C05484=1159.345,41.172,-49.319,-179.753,6.177,149.041
C05485=1159.351,40.923,-49.303,-179.756,6.176,149.042
C05486=1159.355,40.674,-49.288,-179.758,6.176,149.043
C05487=1159.361,40.424,-49.273,-179.761,6.174,149.043
C05488=1159.365,40.174,-49.258,-179.763,6.173,149.044
C05489=1159.371,39.924,-49.242,-179.766,6.173,149.044
C05490=1159.375,39.675,-49.227,-179.769,6.171,149.045
C05491=1159.381,39.425,-49.212,-179.771,6.171,149.045
C05492=1159.386,39.176,-49.198,-179.774,6.170,149.046
C05493=1159.391,38.927,-49.182,-179.777,6.169,149.047
C05494=1159.396,38.678,-49.167,-179.779,6.168,149.047
C05495=1159.401,38.428,-49.152,-179.782,6.167,149.048
C05496=1159.405,38.178,-49.137,-179.784,6.166,149.048
C05497=1159.411,37.928,-49.121,-179.787,6.165,149.049
C05498=1159.415,37.679,-49.106,-179.789,6.164,149.049
C05499=1159.421,37.429,-49.091,-179.792,6.163,149.050
C05500=1159.426,37.180,-49.076,-179.795,6.162,149.050
C05501=1159.431,36.931,-49.061,-179.797,6.162,149.051
C05502=1159.436,36.681,-49.046,-179.800,6.160,149.052
C05503=1159.441,36.432,-49.031,-179.803,6.160,149.052
C05504=1159.446,36.183,-49.016,-179.805,6.159,149.053
C05505=1159.452,35.933,-49.001,-179.807,6.158,149.053
C05506=1159.456,35.684,-48.986,-179.810,6.157,149.054
C05507=1159.462,35.434,-48.970,-179.813,6.156,149.054
C05508=1159.466,35.184,-48.956,-179.815,6.155,149.055
C05509=1159.471,34.935,-48.941,-179.818,6.154,149.056
C05510=1159.477,34.685,-48.926,-179.820,6.153,149.056
C05511=1159.481,34.436,-48.911,-179.823,6.153,149.057
C05512=1159.487,34.186,-48.895,-179.826,6.151,149.057
C05513=1159.491,33.936,-48.881,-179.828,6.151,149.058
C05514=1159.496,33.687,-48.866,-179.831,6.150,149.058
C05515=1159.502,33.437,-48.851,-179.834,6.148,149.059
C05516=1159.506,33.188,-48.836,-179.836,6.148,149.059
C05517=1159.511,32.939,-48.822,-179.839,6.147,149.060
C05518=1159.517,32.689,-48.806,-179.841,6.146,149.061
C05519=1159.522,32.439,-48.792,-179.844,6.145,149.061
C05520=1159.526,32.190,-48.777,-179.846,6.144,149.062
C05521=1159.532,31.941,-48.761,-179.849,6.144,149.062
C05522=1159.537,31.691,-48.747,-179.852,6.142,149.063
C05523=1159.542,31.441,-48.733,-179.854,6.142,149.063
C05524=1159.547,31.192,-48.717,-179.856,6.141,149.064
C05525=1159.552,30.942,-48.703,-179.859,6.140,149.065
C05526=1159.557,30.693,-48.688,-179.862,6.139,149.065
C05527=1159.562,30.443,-48.673,-179.864,6.138,149.066
C05528=1159.567,30.194,-48.658,-179.867,6.137,149.066
C05529=1159.572,29.944,-48.644,-179.870,6.136,149.067
C05530=1159.577,29.695,-48.628,-179.872,6.135,149.067
C05531=1159.582,29.445,-48.614,-179.875,6.135,149.068
C05532=1159.587,29.196,-48.600,-179.877,6.134,149.068
C05533=1159.592,28.947,-48.585,-179.880,6.133,149.069
C05534=1159.598,28.697,-48.570,-179.882,6.132,149.070
C05535=1159.602,28.447,-48.555,-179.885,6.131,149.070
C05536=1159.608,28.178,-48.540,-179.888,6.130,149.071
C05537=1159.613,27.910,-48.525,-179.890,6.129,149.071
C05538=1159.619,27.641,-48.508,-179.893,6.129,149.072
C05539=1159.624,27.372,-48.493,-179.896,6.127,149.073
C05540=1159.629,27.122,-48.478,-179.898,6.127,149.073
C05541=1159.635,26.873,-48.463,-179.901,6.126,149.074
C05542=1159.640,26.623,-48.448,-179.904,6.125,149.074
C05543=1159.645,26.373,-48.434,-179.906,6.124,149.075
C05544=1159.649,26.124,-48.419,-179.909,6.123,149.075
C05545=1159.654,25.875,-48.405,-179.911,6.123,149.076
C05546=1159.659,25.625,-48.391,-179.914,6.121,149.077
C05547=1159.665,25.375,-48.376,-179.917,6.121,149.077
C05548=1159.670,25.127,-48.361,-179.919,6.120,149.078
C05549=1159.675,24.877,-48.347,-179.921,6.119,149.078
C05550=1159.680,24.627,-48.332,-179.924,6.118,149.079
C05551=1159.685,24.377,-48.318,-179.927,6.117,149.080
C05552=1159.690,24.128,-48.303,-179.929,6.116,149.080
C05553=1159.695,23.878,-48.288,-179.932,6.116,149.081
C05554=1159.700,23.629,-48.274,-179.934,6.114,149.081
C05555=1159.705,23.379,-48.260,-179.937,6.114,149.082
C05556=1159.711,23.130,-48.246,-179.939,6.113,149.082
C05557=1159.716,22.881,-48.231,-179.942,6.112,149.083
C05558=1159.720,22.631,-48.217,-179.945,6.111,149.083
C05559=1159.725,22.381,-48.202,-179.947,6.110,149.084
C05560=1159.730,22.132,-48.188,-179.949,6.110,149.084
C05561=1159.735,21.882,-48.174,-179.952,6.109,149.085
C05562=1159.741,21.633,-48.160,-179.954,6.108,149.086
C05563=1159.746,21.384,-48.144,-179.958,6.107,149.086
C05564=1159.751,21.134,-48.130,-179.960,6.106,149.087
C05565=1159.756,20.884,-48.116,-179.962,6.106,149.087
C05566=1159.761,20.634,-48.101,-179.964,6.105,149.088
C05567=1159.766,20.385,-48.087,-179.968,6.104,149.089
C05568=1159.772,20.136,-48.073,-179.970,6.103,149.089
C05569=1159.777,19.886,-48.059,-179.973,6.102,149.090
C05570=1159.782,19.636,-48.045,-179.975,6.102,149.090
C05571=1159.787,19.387,-48.030,-179.977,6.101,149.091
C05572=1159.791,19.137,-48.016,-179.981,6.100,149.092
C05573=1159.797,18.888,-48.002,-179.983,6.099,149.092
C05574=1159.802,18.638,-47.988,-179.985,6.098,149.093
C05575=1159.807,18.388,-47.974,-179.988,6.098,149.093
C05576=1159.812,18.139,-47.959,-179.990,6.097,149.094
C05577=1159.817,17.889,-47.945,-179.993,6.095,149.094
C05578=1159.822,17.640,-47.931,-179.996,6.095,149.095
C05579=1159.827,17.390,-47.917,-179.998,6.094,149.095
C05580=1159.832,17.141,-47.903,180.000,6.094,149.096
C05581=1159.837,16.891,-47.888,179.997,6.093,149.097
C05582=1159.843,16.642,-47.874,179.994,6.092,149.097
C05583=1159.848,16.392,-47.860,179.992,6.091,149.098
C05584=1159.853,16.142,-47.846,179.989,6.090,149.098
C05585=1159.858,15.893,-47.832,179.987,6.089,149.099
C05586=1159.863,15.644,-47.818,179.984,6.089,149.100
C05587=1159.867,15.394,-47.804,179.981,6.088,149.100
C05588=1159.872,15.145,-47.790,179.979,6.087,149.101
C05589=1159.878,14.896,-47.776,179.976,6.086,149.101
C05590=1159.883,14.646,-47.762,179.974,6.086,149.102
C05591=1159.888,14.396,-47.748,179.972,6.085,149.102
C05592=1159.893,14.146,-47.734,179.969,6.084,149.103
C05593=1159.899,13.897,-47.720,179.966,6.083,149.104
C05594=1159.904,13.647,-47.706,179.964,6.082,149.104
C05595=1159.909,13.397,-47.691,179.961,6.082,149.105
C05596=1159.913,13.149,-47.678,179.959,6.081,149.105
C05597=1159.918,12.899,-47.664,179.957,6.080,149.106
C05598=1159.924,12.649,-47.650,179.954,6.079,149.106
C05599=1159.929,12.400,-47.636,179.951,6.078,149.107
C05600=1159.934,12.150,-47.622,179.949,6.078,149.108
C05601=1159.939,11.900,-47.608,179.946,6.077,149.108
C05602=1159.943,11.651,-47.594,179.944,6.076,149.109
C05603=1159.949,11.401,-47.581,179.942,6.076,149.109
C05604=1159.954,11.152,-47.567,179.938,6.075,149.110
C05605=1159.960,10.903,-47.553,179.936,6.074,149.110
C05606=1159.965,10.653,-47.538,179.933,6.073,149.111
C05607=1159.970,10.402,-47.525,179.931,6.072,149.112
C05608=1159.975,10.154,-47.511,179.929,6.072,149.112
C05609=1159.980,9.904,-47.497,179.926,6.071,149.113
C05610=1159.985,9.654,-47.483,179.924,6.071,149.113
C05611=1159.991,9.405,-47.470,179.921,6.069,149.114
C05612=1159.995,9.155,-47.456,179.918,6.069,149.115
C05613=1160.000,8.906,-47.442,179.916,6.068,149.115
C05614=1160.006,8.656,-47.429,179.914,6.067,149.116
C05615=1160.010,8.406,-47.414,179.911,6.066,149.116
C05616=1160.015,8.158,-47.401,179.909,6.066,149.117
C05617=1160.021,7.907,-47.387,179.906,6.066,149.118
C05618=1160.026,7.658,-47.373,179.903,6.064,149.118
C05619=1160.031,7.409,-47.359,179.901,6.064,149.119
C05620=1160.036,7.158,-47.346,179.898,6.063,149.119
C05621=1160.041,6.909,-47.332,179.896,6.062,149.120
C05622=1160.046,6.659,-47.319,179.894,6.061,149.120
C05623=1160.051,6.409,-47.304,179.891,6.061,149.121
C05624=1160.056,6.161,-47.291,179.889,6.060,149.121
C05625=1160.061,5.910,-47.278,179.886,6.059,149.122
C05626=1160.067,5.661,-47.264,179.883,6.058,149.123
C05627=1160.072,5.411,-47.251,179.881,6.058,149.123
C05628=1160.076,5.162,-47.236,179.879,6.057,149.124
C05629=1160.082,4.913,-47.223,179.876,6.056,149.124
C05630=1160.087,4.663,-47.210,179.873,6.056,149.125
C05631=1160.092,4.414,-47.196,179.871,6.055,149.126
C05632=1160.097,4.163,-47.182,179.868,6.055,149.126
C05633=1160.102,3.915,-47.169,179.866,6.053,149.127
C05634=1160.107,3.664,-47.155,179.863,6.052,149.127
C05635=1160.112,3.416,-47.142,179.861,6.052,149.128
C05636=1160.118,3.165,-47.128,179.858,6.051,149.129
C05637=1160.123,2.916,-47.114,179.856,6.050,149.129
C05638=1160.128,2.666,-47.101,179.853,6.050,149.130
C05639=1160.133,2.417,-47.087,179.851,6.049,149.130
C05640=1160.139,2.147,-47.073,179.849,6.049,149.131
C05641=1160.144,1.878,-47.059,179.845,6.047,149.132
C05642=1160.149,1.609,-47.044,179.843,6.047,149.132
C05643=1160.155,1.339,-47.030,179.840,6.046,149.133
C05644=1160.160,1.090,-47.016,179.838,6.046,149.133
C05645=1160.165,0.840,-47.003,179.836,6.045,149.134
C05646=1160.170,0.591,-46.989,179.832,6.044,149.135
C05647=1160.176,0.341,-46.976,179.830,6.043,149.135
C05648=1160.181,0.091,-46.963,179.828,6.042,149.136
C05649=1160.186,-0.158,-46.949,179.825,6.042,149.136
C05650=1160.191,-0.408,-46.936,179.823,6.041,149.137
C05651=1160.196,-0.657,-46.923,179.820,6.041,149.138
C05652=1160.201,-0.907,-46.909,179.818,6.040,149.138
C05653=1160.207,-1.157,-46.896,179.815,6.039,149.139
C05654=1160.211,-1.407,-46.883,179.813,6.039,149.139
C05655=1160.217,-1.656,-46.869,179.810,6.038,149.140
C05656=1160.221,-1.906,-46.856,179.808,6.037,149.140
C05657=1160.227,-2.155,-46.843,179.805,6.036,149.141
C05658=1160.231,-2.405,-46.829,179.802,6.036,149.142
C05659=1160.237,-2.654,-46.816,179.800,6.035,149.142
C05660=1160.242,-2.904,-46.803,179.798,6.034,149.143
C05661=1160.247,-3.153,-46.789,179.795,6.033,149.143
C05662=1160.253,-3.403,-46.776,179.793,6.033,149.144
C05663=1160.257,-3.653,-46.763,179.791,6.032,149.144
C05664=1160.263,-3.902,-46.750,179.788,6.032,149.145
C05665=1160.267,-4.152,-46.736,179.786,6.031,149.146
C05666=1160.273,-4.401,-46.723,179.783,6.031,149.146
C05667=1160.278,-4.651,-46.711,179.781,6.030,149.147
C05668=1160.283,-4.901,-46.697,179.778,6.029,149.147
C05669=1160.288,-5.150,-46.684,179.776,6.028,149.148
C05670=1160.293,-5.400,-46.670,179.773,6.028,149.149
C05671=1160.299,-5.649,-46.658,179.770,6.027,149.149
C05672=1160.304,-5.899,-46.645,179.768,6.026,149.150
C05673=1160.309,-6.149,-46.631,179.765,6.025,149.150
C05674=1160.314,-6.398,-46.619,179.763,6.025,149.151
C05675=1160.320,-6.647,-46.605,179.760,6.024,149.152
C05676=1160.324,-6.897,-46.592,179.758,6.023,149.152
C05677=1160.329,-7.147,-46.579,179.756,6.023,149.153
C05678=1160.335,-7.397,-46.566,179.753,6.022,149.153
C05679=1160.340,-7.646,-46.553,179.751,6.022,149.154
C05680=1160.345,-7.896,-46.541,179.749,6.021,149.154
C05681=1160.350,-8.146,-46.527,179.746,6.020,149.155
C05682=1160.355,-8.395,-46.514,179.743,6.020,149.156
C05683=1160.360,-8.644,-46.501,179.741,6.019,149.156
C05684=1160.365,-8.894,-46.488,179.738,6.019,149.157
C05685=1160.370,-9.144,-46.475,179.736,6.018,149.157
C05686=1160.376,-9.393,-46.462,179.734,6.017,149.158
C05687=1160.381,-9.643,-46.449,179.731,6.017,149.159
C05688=1160.386,-9.893,-46.436,179.729,6.016,149.159
C05689=1160.391,-10.142,-46.424,179.727,6.015,149.160
C05690=1160.396,-10.392,-46.410,179.724,6.015,149.160
C05691=1160.401,-10.642,-46.397,179.722,6.014,149.161
C05692=1160.407,-10.891,-46.385,179.719,6.014,149.162
C05693=1160.412,-11.141,-46.371,179.716,6.012,149.162
C05694=1160.417,-11.391,-46.359,179.714,6.012,149.163
C05695=1160.422,-11.640,-46.346,179.711,6.011,149.163
C05696=1160.427,-11.890,-46.333,179.709,6.010,149.164
C05697=1160.432,-12.140,-46.320,179.706,6.010,149.165
C05698=1160.438,-12.389,-46.307,179.704,6.009,149.165
C05699=1160.443,-12.638,-46.295,179.701,6.009,149.166
C05700=1160.447,-12.888,-46.282,179.699,6.008,149.166
C05701=1160.453,-13.138,-46.269,179.697,6.007,149.167
C05702=1160.458,-13.387,-46.256,179.694,6.007,149.167
C05703=1160.463,-13.637,-46.243,179.692,6.006,149.168
C05704=1160.468,-13.887,-46.230,179.689,6.006,149.169
C05705=1160.473,-14.136,-46.218,179.687,6.005,149.169
C05706=1160.479,-14.385,-46.205,179.684,6.004,149.170
C05707=1160.484,-14.636,-46.192,179.682,6.004,149.170
C05708=1160.489,-14.885,-46.180,179.679,6.003,149.171
C05709=1160.494,-15.135,-46.167,179.677,6.002,149.172
C05710=1160.499,-15.384,-46.155,179.675,6.002,149.172
C05711=1160.504,-15.634,-46.141,179.672,6.001,149.173
C05712=1160.509,-15.884,-46.128,179.670,6.001,149.173
C05713=1160.515,-16.133,-46.116,179.668,6.000,149.174
C05714=1160.520,-16.382,-46.103,179.665,5.999,149.175
C05715=1160.525,-16.632,-46.091,179.662,5.999,149.175
C05716=1160.530,-16.882,-46.078,179.660,5.998,149.176
C05717=1160.535,-17.132,-46.065,179.657,5.998,149.176
C05718=1160.541,-17.381,-46.053,179.655,5.997,149.177
C05719=1160.546,-17.631,-46.040,179.653,5.997,149.178
C05720=1160.551,-17.881,-46.028,179.650,5.996,149.178
C05721=1160.556,-18.131,-46.015,179.648,5.995,149.179
C05722=1160.561,-18.380,-46.002,179.646,5.994,149.179
C05723=1160.566,-18.629,-45.990,179.643,5.994,149.180
C05724=1160.572,-18.879,-45.977,179.641,5.993,149.180
C05725=1160.577,-19.129,-45.965,179.638,5.993,149.181
C05726=1160.582,-19.379,-45.952,179.635,5.992,149.182
C05727=1160.587,-19.628,-45.939,179.633,5.992,149.182
C05728=1160.592,-19.877,-45.927,179.631,5.991,149.183
C05729=1160.597,-20.127,-45.915,179.628,5.990,149.183
C05730=1160.603,-20.377,-45.902,179.626,5.990,149.184
C05731=1160.608,-20.626,-45.890,179.624,5.989,149.185
C05732=1160.613,-20.877,-45.877,179.621,5.989,149.185
C05733=1160.618,-21.126,-45.865,179.619,5.988,149.186
C05734=1160.623,-21.375,-45.852,179.616,5.987,149.186
C05735=1160.628,-21.625,-45.840,179.614,5.987,149.187
C05736=1160.633,-21.874,-45.828,179.612,5.987,149.188
C05737=1160.638,-22.124,-45.815,179.609,5.987,149.188
C05738=1160.645,-22.374,-45.803,179.607,5.986,149.189
C05739=1160.649,-22.624,-45.790,179.604,5.985,149.189
C05740=1160.654,-22.873,-45.777,179.602,5.984,149.190
C05741=1160.660,-23.123,-45.765,179.599,5.984,149.191
C05742=1160.665,-23.373,-45.752,179.597,5.983,149.191
C05743=1160.670,-23.623,-45.741,179.595,5.983,149.192
C05744=1160.675,-23.892,-45.727,179.592,5.982,149.193
C05745=1160.681,-24.162,-45.714,179.590,5.982,149.193
C05746=1160.686,-24.432,-45.701,179.586,5.980,149.194
C05747=1160.692,-24.702,-45.687,179.584,5.980,149.194
C05748=1160.697,-24.952,-45.674,179.582,5.979,149.195
C05749=1160.703,-25.202,-45.663,179.579,5.979,149.196
C05750=1160.708,-25.451,-45.650,179.577,5.978,149.196
C05751=1160.713,-25.700,-45.637,179.575,5.978,149.197
C05752=1160.718,-25.950,-45.625,179.573,5.977,149.197
C05753=1160.723,-26.199,-45.613,179.570,5.977,149.198
C05754=1160.728,-26.449,-45.602,179.567,5.977,149.199
C05755=1160.733,-26.698,-45.589,179.565,5.976,149.199
C05756=1160.739,-26.948,-45.577,179.562,5.975,149.200
C05757=1160.744,-27.198,-45.565,179.560,5.975,149.200
C05758=1160.749,-27.448,-45.552,179.558,5.974,149.201
C05759=1160.754,-27.698,-45.540,179.555,5.973,149.201
C05760=1160.759,-27.948,-45.528,179.553,5.973,149.202
C05761=1160.764,-28.197,-45.515,179.551,5.972,149.203
C05762=1160.770,-28.447,-45.503,179.548,5.972,149.203
C05763=1160.775,-28.697,-45.491,179.546,5.971,149.204
C05764=1160.780,-28.946,-45.479,179.543,5.970,149.204
C05765=1160.785,-29.196,-45.468,179.541,5.970,149.205
C05766=1160.790,-29.445,-45.455,179.538,5.969,149.206
C05767=1160.796,-29.695,-45.443,179.536,5.970,149.206
C05768=1160.801,-29.944,-45.430,179.534,5.969,149.207
C05769=1160.806,-30.194,-45.419,179.531,5.968,149.207
C05770=1160.812,-30.444,-45.407,179.529,5.968,149.208
C05771=1160.816,-30.693,-45.395,179.526,5.967,149.209
C05772=1160.821,-30.943,-45.383,179.524,5.966,149.209
C05773=1160.827,-31.192,-45.370,179.522,5.966,149.210
C05774=1160.832,-31.442,-45.358,179.519,5.965,149.210
C05775=1160.837,-31.692,-45.346,179.517,5.965,149.211
C05776=1160.842,-31.941,-45.334,179.515,5.964,149.211
C05777=1160.847,-32.191,-45.323,179.512,5.963,149.212
C05778=1160.853,-32.441,-45.311,179.510,5.963,149.213
C05779=1160.858,-32.690,-45.298,179.508,5.963,149.213
C05780=1160.863,-32.940,-45.286,179.505,5.963,149.214
C05781=1160.868,-33.190,-45.275,179.503,5.962,149.214
C05782=1160.873,-33.440,-45.263,179.500,5.961,149.215
C05783=1160.878,-33.689,-45.250,179.498,5.961,149.216
C05784=1160.884,-33.939,-45.238,179.495,5.960,149.216
C05785=1160.889,-34.189,-45.227,179.493,5.959,149.217
C05786=1160.894,-34.438,-45.215,179.490,5.959,149.218
C05787=1160.899,-34.688,-45.203,179.488,5.958,149.218
C05788=1160.905,-34.937,-45.191,179.486,5.958,149.219
C05789=1160.911,-35.187,-45.179,179.483,5.957,149.219
C05790=1160.915,-35.436,-45.167,179.481,5.957,149.220
C05791=1160.920,-35.686,-45.155,179.479,5.956,149.220
C05792=1160.926,-35.936,-45.144,179.476,5.956,149.221
C05793=1160.931,-36.186,-45.132,179.474,5.955,149.222
C05794=1160.936,-36.436,-45.120,179.472,5.955,149.222
C05795=1160.941,-36.685,-45.108,179.469,5.954,149.223
C05796=1160.947,-36.935,-45.096,179.467,5.954,149.223
C05797=1160.951,-37.185,-45.085,179.464,5.953,149.224
C05798=1160.957,-37.435,-45.073,179.462,5.952,149.225
C05799=1160.962,-37.684,-45.061,179.460,5.953,149.225
C05800=1160.967,-37.933,-45.049,179.458,5.952,149.226
C05801=1160.972,-38.183,-45.037,179.455,5.951,149.226
C05802=1160.978,-38.433,-45.025,179.453,5.951,149.227
C05803=1160.983,-38.682,-45.014,179.450,5.950,149.228
C05804=1160.988,-38.932,-45.002,179.448,5.949,149.228
C05805=1160.993,-39.182,-44.990,179.445,5.949,149.229
C05806=1160.998,-39.432,-44.979,179.443,5.948,149.229
C05807=1161.004,-39.682,-44.967,179.441,5.949,149.230
C05808=1161.009,-39.932,-44.955,179.439,5.948,149.230
C05809=1161.014,-40.180,-44.944,179.436,5.947,149.231
C05810=1161.019,-40.430,-44.932,179.434,5.947,149.232
C05811=1161.025,-40.680,-44.920,179.431,5.946,149.232
C05812=1161.030,-40.929,-44.909,179.429,5.945,149.233
C05813=1161.035,-41.179,-44.897,179.427,5.945,149.233
C05814=1161.040,-41.429,-44.885,179.424,5.944,149.234
C05815=1161.046,-41.678,-44.874,179.422,5.945,149.235
C05816=1161.051,-41.928,-44.862,179.420,5.944,149.235
C05817=1161.056,-42.178,-44.851,179.417,5.943,149.236
C05818=1161.061,-42.428,-44.839,179.415,5.943,149.237
C05819=1161.066,-42.677,-44.828,179.413,5.942,149.237
C05820=1161.071,-42.927,-44.816,179.410,5.942,149.238
C05821=1161.077,-43.176,-44.805,179.408,5.941,149.238
C05822=1161.082,-43.426,-44.793,179.406,5.941,149.239
C05823=1161.088,-43.676,-44.781,179.403,5.941,149.239
C05824=1161.092,-43.926,-44.770,179.401,5.940,149.240
C05825=1161.098,-44.176,-44.758,179.399,5.939,149.241
C05826=1161.102,-44.425,-44.746,179.396,5.939,149.241
C05827=1161.108,-44.675,-44.735,179.394,5.938,149.242
C05828=1161.113,-44.924,-44.724,179.391,5.938,149.242
C05829=1161.118,-45.174,-44.712,179.390,5.938,149.243
C05830=1161.123,-45.424,-44.700,179.387,5.937,149.244
C05831=1161.129,-45.674,-44.689,179.385,5.936,149.244
C05832=1161.134,-45.923,-44.678,179.382,5.936,149.245
C05833=1161.140,-46.173,-44.667,179.380,5.935,149.245
C05834=1161.144,-46.423,-44.655,179.377,5.935,149.246
C05835=1161.150,-46.673,-44.643,179.376,5.935,149.246
C05836=1161.155,-46.922,-44.632,179.373,5.934,149.247
C05837=1161.160,-47.172,-44.621,179.371,5.934,149.248
C05838=1161.165,-47.421,-44.609,179.368,5.933,149.248
C05839=1161.171,-47.671,-44.597,179.366,5.932,149.249
C05840=1161.176,-47.920,-44.586,179.363,5.932,149.249
C05841=1161.182,-48.171,-44.575,179.362,5.932,149.250
C05842=1161.186,-48.420,-44.564,179.359,5.932,149.251
C05843=1161.192,-48.670,-44.552,179.356,5.931,149.251
C05844=1161.197,-48.919,-44.541,179.354,5.930,149.252
C05845=1161.202,-49.169,-44.530,179.351,5.930,149.253
C05846=1161.207,-49.419,-44.518,179.349,5.929,149.253
C05847=1161.212,-49.669,-44.507,179.347,5.930,149.254
C05848=1161.218,-49.939,-44.495,179.345,5.929,149.254
C05849=1161.224,-50.210,-44.483,179.342,5.928,149.255
C05850=1161.230,-50.480,-44.471,179.340,5.928,149.256
C05851=1161.236,-50.751,-44.458,179.337,5.927,149.256
C05852=1161.240,-51.000,-44.447,179.335,5.927,149.257
C05853=1161.246,-51.250,-44.436,179.333,5.926,149.257
C05854=1161.251,-51.499,-44.424,179.330,5.926,149.258
C05855=1161.256,-51.750,-44.414,179.328,5.926,149.258
C05856=1161.261,-51.999,-44.402,179.326,5.925,149.259
C05857=1161.267,-52.248,-44.391,179.323,5.924,149.260
C05858=1161.271,-52.498,-44.380,179.321,5.924,149.260
C05859=1161.277,-52.749,-44.368,179.319,5.923,149.261
C05860=1161.282,-52.997,-44.358,179.316,5.923,149.262
C05861=1161.287,-53.247,-44.346,179.314,5.923,149.262
C05862=1161.293,-53.498,-44.335,179.312,5.922,149.263
C05863=1161.298,-53.747,-44.324,179.310,5.922,149.263
C05864=1161.303,-53.996,-44.313,179.307,5.921,149.264
C05865=1161.309,-54.247,-44.302,179.305,5.920,149.264
C05866=1161.314,-54.496,-44.291,179.303,5.921,149.265
C05867=1161.319,-54.745,-44.279,179.300,5.920,149.266
C05868=1161.324,-54.996,-44.268,179.298,5.920,149.266
C05869=1161.330,-55.245,-44.257,179.296,5.919,149.267
C05870=1161.334,-55.494,-44.246,179.293,5.918,149.267
C05871=1161.340,-55.745,-44.235,179.291,5.918,149.268
C05872=1161.345,-55.994,-44.224,179.289,5.918,149.269
C05873=1161.350,-56.244,-44.213,179.286,5.917,149.269
C05874=1161.355,-56.494,-44.202,179.284,5.917,149.270
C05875=1161.361,-56.743,-44.191,179.282,5.917,149.270
C05876=1161.366,-56.993,-44.180,179.280,5.916,149.271
C05877=1161.371,-57.242,-44.169,179.277,5.916,149.271
C05878=1161.376,-57.492,-44.159,179.275,5.915,149.272
C05879=1161.382,-57.742,-44.147,179.272,5.914,149.273
C05880=1161.387,-57.992,-44.136,179.270,5.915,149.273
C05881=1161.392,-58.242,-44.125,179.268,5.914,149.274
C05882=1161.397,-58.491,-44.114,179.266,5.914,149.275
C05883=1161.403,-58.741,-44.103,179.263,5.913,149.275
C05884=1161.408,-58.991,-44.092,179.261,5.912,149.276
C05885=1161.413,-59.240,-44.082,179.259,5.912,149.276
C05886=1161.418,-59.490,-44.070,179.256,5.912,149.277
C05887=1161.423,-59.740,-44.060,179.254,5.911,149.277
C05888=1161.429,-59.989,-44.048,179.252,5.911,149.278
C05889=1161.434,-60.240,-44.038,179.250,5.911,149.279
C05890=1161.439,-60.488,-44.027,179.247,5.910,149.279
C05891=1161.444,-60.739,-44.016,179.245,5.910,149.280
C05892=1161.450,-60.988,-44.005,179.242,5.909,149.280
C05893=1161.455,-61.238,-43.994,179.241,5.909,149.281
C05894=1161.460,-61.488,-43.983,179.238,5.909,149.282
C05895=1161.466,-61.737,-43.973,179.236,5.908,149.282
C05896=1161.471,-61.988,-43.962,179.233,5.908,149.283
C05897=1161.476,-62.237,-43.951,179.231,5.907,149.283
C05898=1161.481,-62.487,-43.940,179.229,5.907,149.284
C05899=1161.486,-62.736,-43.930,179.227,5.906,149.284
C05900=1161.492,-62.986,-43.918,179.224,5.906,149.285
C05901=1161.498,-63.236,-43.908,179.222,5.905,149.286
C05902=1161.502,-63.485,-43.897,179.220,5.906,149.286
C05903=1161.508,-63.735,-43.887,179.218,5.905,149.287
C05904=1161.513,-63.985,-43.875,179.215,5.904,149.288
C05905=1161.518,-64.234,-43.865,179.213,5.904,149.288
C05906=1161.523,-64.484,-43.855,179.211,5.904,149.289
C05907=1161.528,-64.734,-43.843,179.209,5.903,149.289
C05908=1161.534,-64.984,-43.832,179.206,5.902,149.290
C05909=1161.539,-65.234,-43.822,179.204,5.902,149.290
C05910=1161.544,-65.483,-43.811,179.202,5.902,149.291
C05911=1161.549,-65.733,-43.800,179.200,5.902,149.292
C05912=1161.555,-65.983,-43.790,179.197,5.901,149.292
C05913=1161.560,-66.232,-43.779,179.195,5.901,149.293
C05914=1161.565,-66.482,-43.769,179.193,5.901,149.293
C05915=1161.571,-66.732,-43.759,179.190,5.900,149.294
C05916=1161.576,-66.981,-43.747,179.188,5.899,149.294
C05917=1161.581,-67.231,-43.737,179.186,5.900,149.295
C05918=1161.586,-67.481,-43.726,179.184,5.899,149.296
C05919=1161.592,-67.730,-43.716,179.181,5.899,149.296
C05920=1161.597,-67.980,-43.705,179.179,5.898,149.297
C05921=1161.602,-68.230,-43.695,179.177,5.898,149.298
C05922=1161.607,-68.480,-43.684,179.175,5.897,149.298
C05923=1161.613,-68.729,-43.674,179.172,5.897,149.299
C05924=1161.617,-68.979,-43.663,179.170,5.896,149.299
C05925=1161.623,-69.229,-43.652,179.168,5.896,149.300
C05926=1161.628,-69.479,-43.642,179.166,5.896,149.300
C05927=1161.634,-69.728,-43.632,179.164,5.895,149.301
C05928=1161.639,-69.977,-43.621,179.161,5.895,149.302
C05929=1161.644,-70.228,-43.610,179.159,5.895,149.302
C05930=1161.649,-70.477,-43.600,179.157,5.894,149.303
C05931=1161.654,-70.727,-43.589,179.154,5.893,149.303
C05932=1161.660,-70.977,-43.579,179.152,5.894,149.304
C05933=1161.665,-71.227,-43.569,179.150,5.893,149.304
C05934=1161.670,-71.476,-43.558,179.147,5.893,149.305
C05935=1161.676,-71.726,-43.547,179.145,5.892,149.306
C05936=1161.681,-71.976,-43.537,179.144,5.892,149.306
C05937=1161.687,-72.225,-43.527,179.141,5.892,149.307
C05938=1161.692,-72.476,-43.516,179.139,5.891,149.307
C05939=1161.697,-72.725,-43.506,179.137,5.891,149.308
C05940=1161.703,-72.975,-43.496,179.135,5.890,149.308
C05941=1161.707,-73.224,-43.484,179.132,5.890,149.309
C05942=1161.713,-73.474,-43.474,179.130,5.889,149.310
C05943=1161.718,-73.724,-43.464,179.128,5.890,149.310
C05944=1161.724,-73.974,-43.453,179.125,5.889,149.311
C05945=1161.729,-74.223,-43.443,179.123,5.888,149.312
C05946=1161.734,-74.473,-43.433,179.121,5.888,149.312
C05947=1161.740,-74.723,-43.422,179.119,5.888,149.312
C05948=1161.745,-74.972,-43.413,179.116,5.887,149.313
C05949=1161.750,-75.222,-43.402,179.115,5.887,149.314
C05950=1161.755,-75.472,-43.392,179.112,5.887,149.314
C05951=1161.761,-75.722,-43.382,179.110,5.886,149.315
C05952=1161.767,-75.993,-43.370,179.107,5.886,149.316
C05953=1161.772,-76.264,-43.359,179.104,5.885,149.316
C05954=1161.778,-76.536,-43.348,179.103,5.885,149.317
C05955=1161.784,-76.807,-43.337,179.100,5.885,149.317
C05956=1161.789,-77.057,-43.327,179.098,5.884,149.318
C05957=1161.794,-77.306,-43.316,179.095,5.884,149.319
C05958=1161.800,-77.556,-43.306,179.094,5.884,149.319
C05959=1161.805,-77.806,-43.296,179.091,5.883,149.320
C05960=1161.810,-78.056,-43.285,179.089,5.883,149.320
C05961=1161.815,-78.305,-43.276,179.087,5.883,149.321
C05962=1161.821,-78.555,-43.266,179.085,5.882,149.322
C05963=1161.826,-78.805,-43.255,179.082,5.881,149.322
C05964=1161.832,-79.054,-43.245,179.080,5.882,149.323
C05965=1161.837,-79.304,-43.235,179.078,5.881,149.323
C05966=1161.841,-79.554,-43.225,179.076,5.881,149.324
C05967=1161.847,-79.803,-43.214,179.074,5.881,149.324
C05968=1161.853,-80.053,-43.204,179.071,5.880,149.325
C05969=1161.858,-80.303,-43.194,179.069,5.880,149.326
C05970=1161.863,-80.553,-43.183,179.067,5.880,149.326
C05971=1161.868,-80.802,-43.174,179.065,5.879,149.327
C05972=1161.874,-81.051,-43.164,179.063,5.878,149.327
C05973=1161.879,-81.302,-43.154,179.060,5.878,149.328
C05974=1161.885,-81.552,-43.144,179.058,5.878,149.328
C05975=1161.889,-81.801,-43.134,179.056,5.877,149.329
C05976=1161.894,-82.051,-43.123,179.053,5.877,149.330
C05977=1161.900,-82.301,-43.113,179.052,5.877,149.330
C05978=1161.906,-82.550,-43.103,179.049,5.876,149.331
C05979=1161.910,-82.800,-43.093,179.047,5.876,149.331
C05980=1161.916,-83.051,-43.083,179.045,5.876,149.332
C05981=1161.921,-83.300,-43.073,179.043,5.875,149.333
C05982=1161.927,-83.550,-43.063,179.041,5.875,149.333
C05983=1161.932,-83.799,-43.053,179.038,5.875,149.334
C05984=1161.937,-84.049,-43.043,179.036,5.874,149.334
C05985=1161.942,-84.299,-43.033,179.034,5.874,149.335
C05986=1161.948,-84.548,-43.024,179.032,5.874,149.335
C05987=1161.953,-84.798,-43.014,179.029,5.873,149.336
C05988=1161.958,-85.048,-43.003,179.028,5.873,149.337
C05989=1161.963,-85.298,-42.993,179.026,5.873,149.337
C05990=1161.969,-85.548,-42.984,179.023,5.872,149.338
C05991=1161.975,-85.797,-42.974,179.021,5.872,149.338
C05992=1161.979,-86.047,-42.964,179.019,5.872,149.339
C05993=1161.984,-86.297,-42.953,179.016,5.871,149.339
C05994=1161.990,-86.547,-42.944,179.015,5.871,149.340
C05995=1161.995,-86.796,-42.934,179.012,5.871,149.341
C05996=1162.001,-87.046,-42.924,179.010,5.870,149.341
C05997=1162.006,-87.296,-42.914,179.008,5.870,149.342
C05998=1162.011,-87.546,-42.905,179.006,5.870,149.342
C05999=1162.017,-87.795,-42.894,179.003,5.869,149.343
C06000=1162.022,-88.045,-42.884,179.001,5.869,149.344
C06001=1162.027,-88.295,-42.875,178.999,5.869,149.344
C06002=1162.032,-88.545,-42.865,178.997,5.868,149.345
C06003=1162.037,-88.794,-42.855,178.995,5.868,149.345
C06004=1162.043,-89.044,-42.845,178.993,5.867,149.346
C06005=1162.049,-89.294,-42.835,178.991,5.868,149.346
C06006=1162.054,-89.543,-42.826,178.989,5.867,149.347
C06007=1162.059,-89.793,-42.816,178.986,5.867,149.348
C06008=1162.064,-90.043,-42.806,178.984,5.867,149.348
C06009=1162.069,-90.293,-42.796,178.982,5.866,149.349
C06010=1162.075,-90.543,-42.787,178.979,5.865,149.349
C06011=1162.080,-90.792,-42.777,178.978,5.866,149.350
C06012=1162.086,-91.042,-42.767,178.975,5.865,149.350
C06013=1162.091,-91.292,-42.758,178.973,5.864,149.351
C06014=1162.096,-91.542,-42.747,178.971,5.864,149.351
C06015=1162.101,-91.792,-42.739,178.969,5.864,149.352
C06016=1162.107,-92.041,-42.728,178.967,5.864,149.353
C06017=1162.112,-92.291,-42.718,178.964,5.864,149.353
C06018=1162.117,-92.541,-42.709,178.962,5.863,149.354
C06019=1162.123,-92.790,-42.699,178.961,5.863,149.354
C06020=1162.128,-93.040,-42.690,178.958,5.863,149.355
C06021=1162.134,-93.289,-42.680,178.956,5.862,149.355
C06022=1162.138,-93.540,-42.671,178.954,5.862,149.356
C06023=1162.144,-93.790,-42.660,178.951,5.861,149.357
C06024=1162.149,-94.039,-42.651,178.950,5.861,149.357
C06025=1162.155,-94.289,-42.641,178.947,5.861,149.358
C06026=1162.159,-94.538,-42.632,178.945,5.860,149.358
C06027=1162.165,-94.788,-42.622,178.943,5.860,149.359
C06028=1162.170,-95.038,-42.613,178.941,5.860,149.360
C06029=1162.176,-95.288,-42.603,178.939,5.860,149.360
C06030=1162.181,-95.537,-42.593,178.937,5.859,149.361
C06031=1162.186,-95.788,-42.584,178.934,5.859,149.361
C06032=1162.191,-96.037,-42.574,178.933,5.859,149.362
C06033=1162.197,-96.287,-42.565,178.930,5.858,149.362
C06034=1162.202,-96.536,-42.555,178.928,5.858,149.363
C06035=1162.208,-96.787,-42.545,178.926,5.858,149.363
C06036=1162.213,-97.037,-42.537,178.924,5.857,149.364
C06037=1162.219,-97.286,-42.526,178.922,5.857,149.365
C06038=1162.224,-97.536,-42.517,178.920,5.857,149.365
C06039=1162.229,-97.785,-42.508,178.917,5.856,149.366
C06040=1162.235,-98.035,-42.498,178.915,5.856,149.366
C06041=1162.239,-98.285,-42.489,178.913,5.855,149.367
C06042=1162.245,-98.535,-42.479,178.911,5.856,149.367
C06043=1162.250,-98.785,-42.470,178.909,5.855,149.368
C06044=1162.256,-99.034,-42.460,178.906,5.855,149.369
C06045=1162.261,-99.284,-42.451,178.905,5.855,149.369
C06046=1162.266,-99.533,-42.442,178.903,5.854,149.370
C06047=1162.272,-99.783,-42.432,178.900,5.854,149.370
C06048=1162.277,-100.033,-42.423,178.898,5.854,149.371
C06049=1162.283,-100.283,-42.413,178.896,5.853,149.371
C06050=1162.287,-100.533,-42.404,178.894,5.853,149.372
C06051=1162.292,-100.783,-42.394,178.892,5.852,149.373
C06052=1162.298,-101.033,-42.385,178.890,5.852,149.373
C06053=1162.303,-101.283,-42.376,178.888,5.852,149.374
C06054=1162.309,-101.532,-42.365,178.886,5.852,149.374
C06055=1162.314,-101.782,-42.357,178.884,5.851,149.375
C06056=1162.320,-102.053,-42.347,178.881,5.851,149.375
C06057=1162.326,-102.325,-42.337,178.879,5.851,149.376
C06058=1162.331,-102.598,-42.327,178.877,5.851,149.377
C06059=1162.338,-102.870,-42.316,178.874,5.850,149.377
C06060=1162.343,-103.119,-42.307,178.872,5.850,149.378
C06061=1162.348,-103.369,-42.298,178.870,5.850,149.378
C06062=1162.354,-103.619,-42.288,178.868,5.849,149.379
C06063=1162.359,-103.869,-42.279,178.866,5.849,149.379
C06064=1162.364,-104.118,-42.270,178.864,5.848,149.380
C06065=1162.370,-104.368,-42.260,178.862,5.849,149.381
C06066=1162.375,-104.618,-42.251,178.860,5.848,149.381
C06067=1162.380,-104.867,-42.242,178.857,5.847,149.382
C06068=1162.385,-105.117,-42.233,178.855,5.848,149.382
C06069=1162.391,-105.367,-42.223,178.853,5.847,149.383
C06070=1162.396,-105.617,-42.214,178.851,5.847,149.383
C06071=1162.401,-105.867,-42.205,178.849,5.847,149.384
C06072=1162.407,-106.117,-42.195,178.847,5.847,149.385
C06073=1162.412,-106.367,-42.186,178.845,5.846,149.385
C06074=1162.417,-106.616,-42.177,178.842,5.846,149.386
C06075=1162.423,-106.866,-42.169,178.841,5.846,149.386
C06076=1162.428,-107.115,-42.159,178.839,5.845,149.387
C06077=1162.433,-107.365,-42.150,178.836,5.845,149.387
C06078=1162.439,-107.615,-42.141,178.834,5.844,149.388
C06079=1162.444,-107.865,-42.132,178.833,5.844,149.388
C06080=1162.450,-108.115,-42.123,178.830,5.844,149.389
C06081=1162.455,-108.365,-42.114,178.828,5.844,149.390
C06082=1162.460,-108.614,-42.104,178.826,5.843,149.390
C06083=1162.465,-108.864,-42.095,178.824,5.843,149.391
C06084=1162.471,-109.114,-42.086,178.822,5.843,149.391
C06085=1162.476,-109.364,-42.077,178.820,5.842,149.392
C06086=1162.481,-109.614,-42.068,178.818,5.842,149.392
C06087=1162.486,-109.863,-42.059,178.815,5.842,149.393
C06088=1162.492,-110.113,-42.050,178.814,5.842,149.393
C06089=1162.498,-110.363,-42.041,178.812,5.841,149.394
C06090=1162.503,-110.613,-42.032,178.810,5.842,149.395
C06091=1162.508,-110.862,-42.022,178.807,5.841,149.395
C06092=1162.513,-111.112,-42.014,178.805,5.840,149.396
C06093=1162.518,-111.362,-42.005,178.803,5.840,149.396
C06094=1162.524,-111.612,-41.995,178.801,5.840,149.397
C06095=1162.529,-111.862,-41.986,178.799,5.840,149.397
C06096=1162.535,-112.111,-41.977,178.797,5.839,149.398
C06097=1162.540,-112.361,-41.969,178.795,5.839,149.399
C06098=1162.545,-112.610,-41.960,178.793,5.839,149.399
C06099=1162.551,-112.860,-41.951,178.791,5.839,149.399
C06100=1162.557,-113.110,-41.941,178.789,5.838,149.400
C06101=1162.562,-113.360,-41.933,178.787,5.838,149.401
C06102=1162.567,-113.610,-41.924,178.785,5.838,149.401
C06103=1162.572,-113.860,-41.915,178.782,5.837,149.402
C06104=1162.578,-114.109,-41.906,178.781,5.837,149.402
C06105=1162.583,-114.359,-41.897,178.778,5.836,149.403
C06106=1162.588,-114.609,-41.888,178.777,5.836,149.403
C06107=1162.594,-114.859,-41.879,178.774,5.836,149.404
C06108=1162.599,-115.109,-41.870,178.772,5.836,149.405
C06109=1162.604,-115.359,-41.861,178.770,5.835,149.405
C06110=1162.610,-115.608,-41.853,178.768,5.836,149.406
C06111=1162.615,-115.858,-41.844,178.766,5.835,149.406
C06112=1162.620,-116.108,-41.835,178.764,5.835,149.407
C06113=1162.626,-116.357,-41.826,178.762,5.834,149.407
C06114=1162.631,-116.607,-41.817,178.760,5.835,149.408
C06115=1162.636,-116.857,-41.808,178.758,5.834,149.408
C06116=1162.642,-117.106,-41.800,178.756,5.834,149.409
C06117=1162.648,-117.356,-41.790,178.754,5.833,149.409
C06118=1162.653,-117.606,-41.781,178.751,5.833,149.410
C06119=1162.658,-117.856,-41.772,178.750,5.833,149.411
C06120=1162.663,-118.107,-41.764,178.748,5.832,149.411
C06121=1162.669,-118.356,-41.756,178.746,5.833,149.412
C06122=1162.674,-118.606,-41.747,178.743,5.832,149.412
C06123=1162.680,-118.855,-41.738,178.742,5.832,149.413
C06124=1162.685,-119.105,-41.729,178.740,5.831,149.413
C06125=1162.690,-119.355,-41.720,178.738,5.832,149.414
C06126=1162.696,-119.604,-41.712,178.735,5.831,149.414
C06127=1162.701,-119.854,-41.703,178.734,5.831,149.415
C06128=1162.706,-120.104,-41.694,178.732,5.830,149.415
C06129=1162.711,-120.354,-41.686,178.729,5.830,149.416
C06130=1162.717,-120.604,-41.677,178.727,5.830,149.417
C06131=1162.722,-120.853,-41.668,178.726,5.830,149.417
C06132=1162.728,-121.103,-41.659,178.723,5.829,149.418
C06133=1162.733,-121.353,-41.650,178.721,5.829,149.418
C06134=1162.738,-121.603,-41.641,178.719,5.829,149.419
C06135=1162.744,-121.853,-41.634,178.718,5.829,149.419
C06136=1162.749,-122.103,-41.625,178.715,5.828,149.420
C06137=1162.754,-122.352,-41.616,178.713,5.828,149.420
C06138=1162.759,-122.602,-41.607,178.711,5.828,149.421
C06139=1162.765,-122.851,-41.598,178.710,5.828,149.421
C06140=1162.771,-123.102,-41.590,178.707,5.827,149.422
C06141=1162.776,-123.352,-41.581,178.705,5.827,149.423
C06142=1162.781,-123.602,-41.572,178.703,5.827,149.423
C06143=1162.787,-123.851,-41.564,178.701,5.827,149.424
C06144=1162.792,-124.101,-41.556,178.699,5.826,149.424
C06145=1162.797,-124.351,-41.547,178.697,5.826,149.425
C06146=1162.803,-124.600,-41.538,178.695,5.826,149.425
C06147=1162.808,-124.850,-41.530,178.693,5.826,149.426
C06148=1162.813,-125.100,-41.522,178.691,5.825,149.426
C06149=1162.818,-125.350,-41.513,178.689,5.825,149.427
C06150=1162.824,-125.599,-41.504,178.687,5.824,149.428
C06151=1162.829,-125.849,-41.495,178.685,5.824,149.428
C06152=1162.835,-126.100,-41.487,178.683,5.824,149.428
C06153=1162.840,-126.349,-41.479,178.682,5.824,149.429
C06154=1162.846,-126.599,-41.470,178.679,5.823,149.430
C06155=1162.851,-126.849,-41.462,178.677,5.823,149.430
C06156=1162.857,-127.098,-41.453,178.675,5.823,149.431
C06157=1162.862,-127.348,-41.444,178.673,5.823,149.431
C06158=1162.867,-127.598,-41.437,178.671,5.822,149.432
C06159=1162.872,-127.848,-41.428,178.669,5.822,149.432
C06160=1162.452,-127.859,-41.469,178.665,5.826,149.434
C06161=1162.446,-127.609,-41.478,178.668,5.826,149.433
C06162=1162.440,-127.359,-41.486,178.670,5.826,149.433
C06163=1162.435,-127.109,-41.495,178.671,5.826,149.433
C06164=1162.430,-126.860,-41.503,178.673,5.827,149.432
C06165=1162.424,-126.610,-41.512,178.675,5.827,149.432
C06166=1162.419,-126.360,-41.520,178.678,5.827,149.431
C06167=1162.414,-126.111,-41.528,178.679,5.827,149.430
C06168=1162.409,-125.861,-41.537,178.681,5.828,149.430
C06169=1162.403,-125.610,-41.545,178.683,5.828,149.429
C06170=1162.397,-125.361,-41.554,178.686,5.828,149.429
C06171=1162.392,-125.111,-41.563,178.687,5.828,149.428
C06172=1162.387,-124.861,-41.571,178.689,5.829,149.428
C06173=1162.382,-124.611,-41.580,178.691,5.829,149.427
C06174=1162.376,-124.362,-41.589,178.693,5.830,149.427
C06175=1162.371,-124.112,-41.597,178.695,5.829,149.426
C06176=1162.365,-123.862,-41.606,178.698,5.830,149.425
C06177=1162.360,-123.612,-41.614,178.699,5.830,149.425
C06178=1162.354,-123.363,-41.623,178.701,5.831,149.425
C06179=1162.349,-123.113,-41.632,178.703,5.830,149.424
C06180=1162.344,-122.863,-41.641,178.706,5.831,149.423
C06181=1162.338,-122.613,-41.649,178.707,5.831,149.423
C06182=1162.333,-122.363,-41.658,178.709,5.832,149.422
C06183=1162.328,-122.114,-41.666,178.712,5.831,149.422
C06184=1162.323,-121.864,-41.675,178.714,5.832,149.421
C06185=1162.317,-121.615,-41.683,178.716,5.833,149.421
C06186=1162.312,-121.364,-41.691,178.717,5.833,149.420
C06187=1162.307,-121.114,-41.700,178.720,5.833,149.419
C06188=1162.302,-120.865,-41.709,178.722,5.833,149.419
C06189=1162.296,-120.615,-41.718,178.724,5.834,149.418
C06190=1162.291,-120.366,-41.727,178.726,5.834,149.418
C06191=1162.285,-120.115,-41.735,178.728,5.834,149.417
C06192=1162.280,-119.865,-41.744,178.730,5.834,149.417
C06193=1162.275,-119.615,-41.753,178.732,5.835,149.416
C06194=1162.268,-119.366,-41.762,178.734,5.835,149.416
C06195=1162.263,-119.116,-41.771,178.736,5.835,149.415
C06196=1162.258,-118.866,-41.780,178.738,5.835,149.415
C06197=1162.253,-118.616,-41.788,178.740,5.836,149.414
C06198=1162.248,-118.367,-41.797,178.742,5.836,149.414
C06199=1162.242,-118.117,-41.806,178.744,5.836,149.413
C06200=1162.236,-117.867,-41.814,178.746,5.836,149.412
C06201=1162.231,-117.617,-41.823,178.748,5.837,149.412
C06202=1162.226,-117.367,-41.832,178.750,5.837,149.411
C06203=1162.221,-117.117,-41.841,178.752,5.837,149.411
C06204=1162.215,-116.868,-41.849,178.754,5.837,149.410
C06205=1162.210,-116.618,-41.858,178.756,5.838,149.410
C06206=1162.205,-116.369,-41.867,178.758,5.838,149.409
C06207=1162.200,-116.119,-41.876,178.761,5.838,149.409
C06208=1162.194,-115.869,-41.885,178.762,5.838,149.408
C06209=1162.188,-115.619,-41.894,178.764,5.839,149.408
C06210=1162.183,-115.370,-41.903,178.767,5.839,149.407
C06211=1162.178,-115.120,-41.912,178.769,5.839,149.406
C06212=1162.172,-114.870,-41.921,178.771,5.840,149.406
C06213=1162.167,-114.620,-41.930,178.772,5.840,149.405
C06214=1162.162,-114.370,-41.939,178.775,5.841,149.405
C06215=1162.156,-114.121,-41.947,178.777,5.840,149.404
C06216=1162.151,-113.871,-41.956,178.779,5.841,149.404
C06217=1162.146,-113.621,-41.965,178.781,5.841,149.403
C06218=1162.140,-113.371,-41.974,178.783,5.842,149.403
C06219=1162.135,-113.121,-41.983,178.785,5.842,149.402
C06220=1162.130,-112.871,-41.992,178.787,5.842,149.402
C06221=1162.125,-112.622,-42.001,178.789,5.842,149.401
C06222=1162.119,-112.372,-42.010,178.791,5.843,149.400
C06223=1162.114,-112.123,-42.018,178.793,5.843,149.400
C06224=1162.108,-111.872,-42.028,178.795,5.843,149.399
C06225=1162.103,-111.623,-42.037,178.798,5.844,149.399
C06226=1162.097,-111.373,-42.046,178.799,5.844,149.398
C06227=1162.092,-111.123,-42.055,178.802,5.844,149.397
C06228=1162.087,-110.873,-42.064,178.804,5.844,149.397
C06229=1162.082,-110.623,-42.072,178.806,5.845,149.396
C06230=1162.076,-110.373,-42.082,178.807,5.845,149.396
C06231=1162.071,-110.124,-42.091,178.810,5.845,149.395
C06232=1162.065,-109.875,-42.100,178.812,5.846,149.395
C06233=1162.060,-109.625,-42.109,178.814,5.846,149.394
C06234=1162.054,-109.375,-42.118,178.816,5.846,149.394
C06235=1162.049,-109.125,-42.127,178.818,5.846,149.393
C06236=1162.044,-108.875,-42.136,178.820,5.847,149.393
C06237=1162.039,-108.625,-42.145,178.822,5.847,149.392
C06238=1162.034,-108.375,-42.154,178.825,5.847,149.391
C06239=1162.028,-108.126,-42.164,178.826,5.847,149.391
C06240=1162.023,-107.876,-42.173,178.829,5.848,149.390
C06241=1162.018,-107.626,-42.182,178.831,5.848,149.390
C06242=1162.013,-107.376,-42.191,178.833,5.848,149.389
C06243=1162.006,-107.127,-42.200,178.835,5.849,149.389
C06244=1162.001,-106.877,-42.209,178.837,5.849,149.388
C06245=1161.996,-106.628,-42.219,178.839,5.850,149.388
C06246=1161.991,-106.378,-42.228,178.841,5.850,149.387
C06247=1161.985,-106.128,-42.237,178.843,5.850,149.386
C06248=1161.980,-105.878,-42.246,178.846,5.851,149.386
C06249=1161.975,-105.628,-42.256,178.847,5.851,149.385
C06250=1161.969,-105.378,-42.265,178.850,5.851,149.385
C06251=1161.964,-105.128,-42.274,178.851,5.851,149.384
C06252=1161.959,-104.879,-42.283,178.854,5.852,149.384
C06253=1161.954,-104.629,-42.292,178.856,5.851,149.383
C06254=1161.948,-104.379,-42.302,178.858,5.852,149.383
C06255=1161.943,-104.129,-42.311,178.860,5.853,149.382
C06256=1161.938,-103.880,-42.320,178.862,5.852,149.381
C06257=1161.932,-103.630,-42.330,178.864,5.853,149.381
C06258=1161.927,-103.380,-42.339,178.866,5.853,149.380
C06259=1161.922,-103.130,-42.348,178.869,5.854,149.380
C06260=1161.916,-102.880,-42.357,178.870,5.854,149.379
C06261=1161.910,-102.608,-42.367,178.873,5.854,149.378
C06262=1161.905,-102.336,-42.378,178.875,5.855,149.378
C06263=1161.899,-102.065,-42.388,178.878,5.855,149.377
C06264=1161.893,-101.793,-42.398,178.879,5.855,149.377
C06265=1161.887,-101.543,-42.407,178.882,5.855,149.376
C06266=1161.882,-101.293,-42.416,178.884,5.855,149.376
C06267=1161.877,-101.044,-42.426,178.886,5.856,149.375
C06268=1161.871,-100.794,-42.435,178.889,5.856,149.374
C06269=1161.866,-100.544,-42.444,178.890,5.856,149.374
C06270=1161.861,-100.294,-42.454,178.892,5.857,149.373
C06271=1161.855,-100.044,-42.463,178.894,5.857,149.373
C06272=1161.851,-99.795,-42.473,178.897,5.858,149.372
C06273=1161.845,-99.545,-42.482,178.899,5.858,149.372
C06274=1161.840,-99.295,-42.491,178.901,5.858,149.371
C06275=1161.834,-99.046,-42.501,178.903,5.859,149.371
C06276=1161.829,-98.795,-42.511,178.905,5.859,149.370
C06277=1161.825,-98.546,-42.520,178.907,5.859,149.369
C06278=1161.819,-98.296,-42.530,178.910,5.860,149.369
C06279=1161.813,-98.046,-42.539,178.911,5.860,149.368
C06280=1161.808,-97.796,-42.549,178.914,5.860,149.368
C06281=1161.803,-97.546,-42.558,178.915,5.860,149.367
C06282=1161.797,-97.297,-42.568,178.918,5.861,149.366
C06283=1161.792,-97.047,-42.577,178.920,5.861,149.366
C06284=1161.786,-96.798,-42.587,178.922,5.861,149.365
C06285=1161.781,-96.548,-42.596,178.925,5.862,149.365
C06286=1161.776,-96.298,-42.605,178.926,5.862,149.364
C06287=1161.770,-96.048,-42.615,178.928,5.862,149.364
C06288=1161.765,-95.798,-42.624,178.931,5.863,149.363
C06289=1161.760,-95.549,-42.634,178.933,5.863,149.363
C06290=1161.754,-95.299,-42.643,178.935,5.864,149.362
C06291=1161.749,-95.049,-42.654,178.937,5.864,149.361
C06292=1161.744,-94.799,-42.663,178.939,5.864,149.361
C06293=1161.739,-94.549,-42.673,178.942,5.864,149.360
C06294=1161.734,-94.300,-42.682,178.943,5.864,149.360
C06295=1161.728,-94.050,-42.692,178.945,5.865,149.359
C06296=1161.723,-93.800,-42.701,178.948,5.865,149.359
C06297=1161.717,-93.551,-42.711,178.950,5.865,149.358
C06298=1161.712,-93.301,-42.721,178.952,5.866,149.358
C06299=1161.706,-93.051,-42.730,178.954,5.866,149.357
C06300=1161.702,-92.802,-42.740,178.956,5.866,149.356
C06301=1161.696,-92.551,-42.750,178.959,5.867,149.356
C06302=1161.691,-92.302,-42.760,178.960,5.867,149.355
C06303=1161.685,-92.052,-42.769,178.963,5.868,149.355
C06304=1161.680,-91.802,-42.779,178.965,5.868,149.354
C06305=1161.675,-91.553,-42.789,178.967,5.868,149.353
C06306=1161.669,-91.303,-42.798,178.970,5.868,149.353
C06307=1161.664,-91.054,-42.808,178.971,5.868,149.352
C06308=1161.659,-90.803,-42.818,178.973,5.869,149.352
C06309=1161.654,-90.553,-42.827,178.976,5.869,149.351
C06310=1161.648,-90.304,-42.837,178.978,5.869,149.351
C06311=1161.643,-90.054,-42.847,178.980,5.870,149.350
C06312=1161.638,-89.805,-42.856,178.983,5.871,149.349
C06313=1161.632,-89.555,-42.867,178.984,5.871,149.349
C06314=1161.628,-89.304,-42.876,178.987,5.871,149.348
C06315=1161.622,-89.055,-42.886,178.989,5.872,149.348
C06316=1161.616,-88.805,-42.896,178.991,5.872,149.347
C06317=1161.611,-88.555,-42.905,178.993,5.872,149.347
C06318=1161.606,-88.306,-42.915,178.995,5.873,149.346
C06319=1161.601,-88.057,-42.925,178.998,5.872,149.345
C06320=1161.595,-87.806,-42.935,179.000,5.873,149.345
C06321=1161.590,-87.556,-42.945,179.001,5.873,149.344
C06322=1161.585,-87.307,-42.955,179.004,5.874,149.344
C06323=1161.579,-87.057,-42.964,179.006,5.874,149.343
C06324=1161.573,-86.807,-42.974,179.008,5.874,149.342
C06325=1161.569,-86.557,-42.984,179.010,5.875,149.342
C06326=1161.564,-86.308,-42.995,179.013,5.876,149.342
C06327=1161.558,-86.058,-43.004,179.015,5.875,149.341
C06328=1161.553,-85.809,-43.014,179.017,5.876,149.340
C06329=1161.548,-85.558,-43.024,179.020,5.876,149.340
C06330=1161.542,-85.309,-43.035,179.021,5.876,149.339
C06331=1161.537,-85.059,-43.043,179.023,5.877,149.339
C06332=1161.531,-84.809,-43.054,179.026,5.877,149.338
C06333=1161.526,-84.559,-43.064,179.028,5.877,149.337
C06334=1161.522,-84.310,-43.074,179.030,5.878,149.337
C06335=1161.516,-84.060,-43.084,179.033,5.879,149.336
C06336=1161.510,-83.810,-43.094,179.035,5.878,149.336
C06337=1161.506,-83.560,-43.103,179.037,5.879,149.335
C06338=1161.500,-83.311,-43.114,179.039,5.880,149.335
C06339=1161.495,-83.061,-43.124,179.041,5.879,149.334
C06340=1161.489,-82.812,-43.134,179.043,5.880,149.333
C06341=1161.485,-82.562,-43.144,179.046,5.880,149.333
C06342=1161.479,-82.311,-43.154,179.048,5.880,149.332
C06343=1161.473,-82.062,-43.164,179.050,5.881,149.332
C06344=1161.468,-81.812,-43.174,179.052,5.882,149.331
C06345=1161.463,-81.562,-43.184,179.054,5.882,149.331
C06346=1161.458,-81.313,-43.194,179.057,5.882,149.330
C06347=1161.452,-81.063,-43.204,179.059,5.883,149.329
C06348=1161.447,-80.814,-43.215,179.061,5.882,149.329
C06349=1161.442,-80.563,-43.224,179.063,5.883,149.328
C06350=1161.436,-80.314,-43.234,179.065,5.884,149.328
C06351=1161.431,-80.064,-43.244,179.067,5.884,149.327
C06352=1161.426,-79.814,-43.255,179.070,5.884,149.326
C06353=1161.420,-79.564,-43.265,179.072,5.885,149.326
C06354=1161.415,-79.315,-43.275,179.074,5.885,149.325
C06355=1161.410,-79.065,-43.285,179.077,5.885,149.325
C06356=1161.405,-78.815,-43.295,179.079,5.886,149.324
C06357=1161.399,-78.566,-43.306,179.080,5.886,149.324
C06358=1161.394,-78.316,-43.316,179.083,5.886,149.323
C06359=1161.389,-78.066,-43.326,179.085,5.887,149.322
C06360=1161.384,-77.817,-43.336,179.087,5.887,149.322
C06361=1161.378,-77.567,-43.346,179.089,5.887,149.321
C06362=1161.373,-77.317,-43.357,179.092,5.888,149.321
C06363=1161.368,-77.067,-43.367,179.094,5.889,149.320
C06364=1161.362,-76.818,-43.377,179.096,5.889,149.320
C06365=1161.357,-76.547,-43.388,179.099,5.889,149.319
C06366=1161.351,-76.275,-43.400,179.101,5.889,149.318
C06367=1161.345,-76.004,-43.410,179.103,5.890,149.318
C06368=1161.339,-75.733,-43.422,179.106,5.890,149.317
C06369=1161.334,-75.483,-43.432,179.108,5.890,149.316
C06370=1161.329,-75.233,-43.443,179.110,5.891,149.316
C06371=1161.324,-74.984,-43.452,179.113,5.892,149.315
C06372=1161.319,-74.734,-43.463,179.115,5.891,149.315
C06373=1161.313,-74.484,-43.473,179.117,5.892,149.314
C06374=1161.308,-74.234,-43.483,179.119,5.892,149.313
C06375=1161.303,-73.984,-43.494,179.122,5.893,149.313
C06376=1161.297,-73.735,-43.504,179.124,5.893,149.312
C06377=1161.291,-73.485,-43.514,179.126,5.894,149.312
C06378=1161.287,-73.236,-43.526,179.128,5.894,149.311
C06379=1161.281,-72.986,-43.536,179.130,5.894,149.311
C06380=1161.276,-72.736,-43.546,179.132,5.895,149.310
C06381=1161.270,-72.486,-43.557,179.135,5.895,149.309
C06382=1161.265,-72.237,-43.567,179.137,5.895,149.309
C06383=1161.260,-71.986,-43.577,179.139,5.895,149.308
C06384=1161.254,-71.737,-43.588,179.142,5.896,149.308
C06385=1161.250,-71.487,-43.598,179.144,5.897,149.307
C06386=1161.245,-71.238,-43.608,179.146,5.897,149.306
C06387=1161.239,-70.988,-43.619,179.148,5.897,149.306
C06388=1161.234,-70.738,-43.629,179.151,5.898,149.305
C06389=1161.228,-70.489,-43.639,179.153,5.899,149.305
C06390=1161.223,-70.238,-43.650,179.155,5.898,149.304
C06391=1161.218,-69.989,-43.660,179.157,5.899,149.304
C06392=1161.213,-69.739,-43.671,179.160,5.899,149.303
C06393=1161.208,-69.490,-43.682,179.161,5.899,149.302
C06394=1161.202,-69.240,-43.692,179.164,5.900,149.302
C06395=1161.197,-68.990,-43.702,179.166,5.901,149.301
C06396=1161.192,-68.741,-43.713,179.169,5.901,149.301
C06397=1161.187,-68.491,-43.724,179.170,5.901,149.300
C06398=1161.181,-68.241,-43.734,179.173,5.901,149.299
C06399=1161.176,-67.991,-43.745,179.175,5.902,149.299
C06400=1161.170,-67.742,-43.756,179.178,5.903,149.298
C06401=1161.165,-67.491,-43.767,179.180,5.903,149.298
C06402=1161.160,-67.242,-43.777,179.182,5.903,149.297
C06403=1161.155,-66.992,-43.788,179.184,5.904,149.296
C06404=1161.149,-66.743,-43.799,179.187,5.904,149.296
C06405=1161.144,-66.493,-43.809,179.189,5.904,149.295
C06406=1161.139,-66.243,-43.819,179.191,5.905,149.295
C06407=1161.133,-65.994,-43.830,179.194,5.905,149.294
C06408=1161.128,-65.744,-43.841,179.195,5.905,149.294
C06409=1161.123,-65.494,-43.851,179.198,5.906,149.293
C06410=1161.118,-65.245,-43.862,179.200,5.906,149.292
C06411=1161.112,-64.995,-43.873,179.203,5.907,149.292
C06412=1161.107,-64.745,-43.883,179.204,5.907,149.291
C06413=1161.102,-64.496,-43.894,179.207,5.907,149.291
C06414=1161.096,-64.245,-43.905,179.209,5.908,149.290
C06415=1161.091,-63.996,-43.915,179.212,5.908,149.289
C06416=1161.086,-63.746,-43.927,179.213,5.908,149.289
C06417=1161.081,-63.496,-43.937,179.216,5.909,149.288
C06418=1161.076,-63.246,-43.948,179.218,5.910,149.288
C06419=1161.071,-62.997,-43.959,179.220,5.910,149.287
C06420=1161.065,-62.747,-43.969,179.223,5.911,149.287
C06421=1161.061,-62.498,-43.980,179.225,5.911,149.286
C06422=1161.054,-62.248,-43.991,179.227,5.911,149.285
C06423=1161.049,-61.998,-44.002,179.230,5.912,149.285
C06424=1161.044,-61.749,-44.013,179.232,5.912,149.284
C06425=1161.039,-61.498,-44.023,179.234,5.912,149.284
C06426=1161.034,-61.249,-44.034,179.237,5.913,149.283
C06427=1161.029,-60.999,-44.045,179.239,5.914,149.282
C06428=1161.023,-60.749,-44.057,179.241,5.914,149.282
C06429=1161.018,-60.500,-44.067,179.243,5.914,149.281
C06430=1161.013,-60.250,-44.078,179.246,5.914,149.281
C06431=1161.007,-60.001,-44.088,179.248,5.915,149.280
C06432=1161.003,-59.751,-44.100,179.250,5.916,149.279
C06433=1160.997,-59.501,-44.110,179.252,5.916,149.279
C06434=1160.992,-59.251,-44.122,179.255,5.916,149.278
C06435=1160.987,-59.001,-44.132,179.257,5.917,149.278
C06436=1160.981,-58.752,-44.143,179.260,5.917,149.277
C06437=1160.976,-58.502,-44.154,179.262,5.918,149.277
C06438=1160.970,-58.253,-44.165,179.264,5.918,149.276
C06439=1160.965,-58.003,-44.176,179.266,5.918,149.275
C06440=1160.961,-57.753,-44.187,179.269,5.919,149.275
C06441=1160.955,-57.503,-44.197,179.271,5.920,149.274
C06442=1160.950,-57.254,-44.209,179.274,5.920,149.273
C06443=1160.945,-57.004,-44.220,179.275,5.920,149.273
C06444=1160.939,-56.754,-44.231,179.278,5.920,149.272
C06445=1160.935,-56.505,-44.242,179.280,5.921,149.272
C06446=1160.928,-56.255,-44.253,179.282,5.922,149.271
C06447=1160.924,-56.005,-44.264,179.284,5.921,149.271
C06448=1160.919,-55.756,-44.275,179.286,5.922,149.270
C06449=1160.913,-55.506,-44.286,179.289,5.923,149.269
C06450=1160.908,-55.256,-44.297,179.291,5.923,149.269
C06451=1160.903,-55.006,-44.308,179.294,5.924,149.268
C06452=1160.898,-54.757,-44.319,179.296,5.924,149.268
C06453=1160.892,-54.507,-44.331,179.298,5.924,149.267
C06454=1160.887,-54.257,-44.341,179.300,5.925,149.267
C06455=1160.882,-54.008,-44.352,179.303,5.925,149.266
C06456=1160.877,-53.758,-44.364,179.305,5.926,149.265
C06457=1160.871,-53.508,-44.375,179.307,5.926,149.265
C06458=1160.866,-53.259,-44.386,179.310,5.927,149.264
C06459=1160.861,-53.009,-44.397,179.312,5.927,149.264
C06460=1160.856,-52.759,-44.408,179.314,5.928,149.263
C06461=1160.850,-52.510,-44.419,179.317,5.928,149.262
C06462=1160.845,-52.260,-44.431,179.319,5.928,149.262
C06463=1160.840,-52.010,-44.442,179.321,5.929,149.261
C06464=1160.835,-51.760,-44.452,179.324,5.929,149.261
C06465=1160.829,-51.511,-44.464,179.326,5.930,149.260
C06466=1160.825,-51.261,-44.476,179.328,5.931,149.260
C06467=1160.820,-51.011,-44.487,179.331,5.931,149.259
C06468=1160.814,-50.761,-44.498,179.333,5.931,149.258
C06469=1160.808,-50.491,-44.511,179.335,5.932,149.258
C06470=1160.802,-50.221,-44.523,179.338,5.932,149.257
C06471=1160.797,-49.950,-44.534,179.341,5.932,149.256
C06472=1160.791,-49.679,-44.547,179.343,5.933,149.256
C06473=1160.785,-49.430,-44.558,179.345,5.934,149.255
C06474=1160.781,-49.180,-44.569,179.348,5.934,149.255
C06475=1160.775,-48.930,-44.581,179.350,5.935,149.254
C06476=1160.770,-48.680,-44.592,179.353,5.936,149.253
C06477=1160.765,-48.431,-44.603,179.355,5.935,149.253
C06478=1160.760,-48.181,-44.615,179.357,5.936,149.252
C06479=1160.755,-47.932,-44.626,179.359,5.936,149.252
C06480=1160.749,-47.682,-44.638,179.362,5.937,149.251
C06481=1160.744,-47.433,-44.649,179.364,5.938,149.250
C06482=1160.739,-47.183,-44.661,179.366,5.938,149.250
C06483=1160.734,-46.933,-44.671,179.369,5.938,149.249
C06484=1160.728,-46.683,-44.683,179.371,5.939,149.249
C06485=1160.723,-46.434,-44.694,179.373,5.939,149.248
C06486=1160.718,-46.184,-44.706,179.376,5.940,149.248
C06487=1160.713,-45.934,-44.717,179.378,5.940,149.247
C06488=1160.707,-45.684,-44.729,179.380,5.941,149.246
C06489=1160.703,-45.435,-44.740,179.383,5.941,149.246
C06490=1160.697,-45.185,-44.752,179.385,5.942,149.245
C06491=1160.692,-44.936,-44.763,179.387,5.942,149.244
C06492=1160.687,-44.686,-44.775,179.390,5.942,149.244
C06493=1160.682,-44.436,-44.786,179.392,5.943,149.243
C06494=1160.676,-44.186,-44.797,179.395,5.944,149.243
C06495=1160.671,-43.937,-44.808,179.397,5.944,149.242
C06496=1160.666,-43.687,-44.820,179.399,5.944,149.241
C06497=1160.661,-43.437,-44.832,179.401,5.945,149.241
C06498=1160.655,-43.187,-44.843,179.404,5.945,149.240
C06499=1160.650,-42.937,-44.855,179.406,5.946,149.240
C06500=1160.645,-42.688,-44.866,179.409,5.946,149.239
C06501=1160.639,-42.438,-44.878,179.411,5.947,149.239
C06502=1160.635,-42.189,-44.889,179.414,5.948,149.238
C06503=1160.629,-41.939,-44.901,179.415,5.948,149.237
C06504=1160.624,-41.689,-44.913,179.418,5.948,149.237
C06505=1160.619,-41.440,-44.925,179.420,5.949,149.236
C06506=1160.613,-41.191,-44.937,179.423,5.949,149.236
C06507=1160.609,-40.941,-44.948,179.425,5.950,149.235
C06508=1160.603,-40.691,-44.960,179.428,5.951,149.234
C06509=1160.598,-40.441,-44.971,179.430,5.951,149.234
C06510=1160.593,-40.192,-44.983,179.432,5.951,149.233
C06511=1160.588,-39.942,-44.995,179.434,5.952,149.233
C06512=1160.583,-39.692,-45.006,179.437,5.952,149.232
C06513=1160.577,-39.443,-45.018,179.439,5.953,149.232
C06514=1160.571,-39.193,-45.030,179.442,5.953,149.231
C06515=1160.567,-38.943,-45.041,179.444,5.954,149.230
C06516=1160.561,-38.693,-45.053,179.446,5.955,149.230
C06517=1160.556,-38.444,-45.065,179.449,5.955,149.229
C06518=1160.552,-38.194,-45.077,179.451,5.955,149.228
C06519=1160.546,-37.944,-45.089,179.453,5.955,149.228
C06520=1160.541,-37.694,-45.101,179.456,5.956,149.227
C06521=1160.535,-37.446,-45.111,179.458,5.957,149.227
C06522=1160.530,-37.196,-45.123,179.460,5.957,149.226
C06523=1160.525,-36.946,-45.136,179.463,5.958,149.225
C06524=1160.520,-36.697,-45.147,179.465,5.959,149.225
C06525=1160.515,-36.447,-45.159,179.468,5.959,149.224
C06526=1160.509,-36.197,-45.171,179.470,5.960,149.224
C06527=1160.504,-35.947,-45.183,179.472,5.960,149.223
C06528=1160.499,-35.698,-45.195,179.474,5.960,149.223
C06529=1160.494,-35.448,-45.207,179.477,5.961,149.222
C06530=1160.489,-35.198,-45.219,179.479,5.962,149.221
C06531=1160.483,-34.948,-45.231,179.482,5.962,149.221
C06532=1160.478,-34.698,-45.242,179.484,5.963,149.220
C06533=1160.473,-34.449,-45.254,179.487,5.963,149.220
C06534=1160.468,-34.199,-45.266,179.489,5.964,149.219
C06535=1160.462,-33.950,-45.278,179.492,5.964,149.218
C06536=1160.457,-33.701,-45.290,179.494,5.965,149.218
C06537=1160.452,-33.451,-45.302,179.496,5.966,149.217
C06538=1160.447,-33.201,-45.314,179.498,5.965,149.217
C06539=1160.441,-32.951,-45.325,179.501,5.966,149.216
C06540=1160.437,-32.702,-45.337,179.503,5.966,149.215
C06541=1160.431,-32.452,-45.349,179.505,5.967,149.215
C06542=1160.426,-32.202,-45.361,179.508,5.968,149.214
C06543=1160.421,-31.953,-45.374,179.510,5.969,149.214
C06544=1160.415,-31.703,-45.386,179.513,5.969,149.213
C06545=1160.411,-31.453,-45.397,179.515,5.970,149.213
C06546=1160.406,-31.204,-45.410,179.518,5.970,149.212
C06547=1160.400,-30.954,-45.422,179.520,5.971,149.211
C06548=1160.395,-30.704,-45.433,179.523,5.971,149.211
C06549=1160.390,-30.455,-45.446,179.525,5.972,149.210
C06550=1160.384,-30.205,-45.458,179.527,5.972,149.210
C06551=1160.380,-29.956,-45.470,179.529,5.973,149.209
C06552=1160.374,-29.706,-45.482,179.532,5.973,149.208
C06553=1160.369,-29.456,-45.494,179.534,5.973,149.208
C06554=1160.364,-29.207,-45.506,179.537,5.974,149.207
C06555=1160.358,-28.957,-45.518,179.539,5.975,149.206
C06556=1160.353,-28.707,-45.531,179.541,5.976,149.206
C06557=1160.348,-28.457,-45.543,179.544,5.976,149.205
C06558=1160.343,-28.208,-45.555,179.546,5.977,149.205
C06559=1160.338,-27.959,-45.567,179.549,5.977,149.204
C06560=1160.333,-27.709,-45.579,179.551,5.978,149.204
C06561=1160.328,-27.459,-45.591,179.554,5.978,149.203
C06562=1160.323,-27.209,-45.604,179.556,5.979,149.202
C06563=1160.317,-26.959,-45.616,179.559,5.980,149.202
C06564=1160.312,-26.710,-45.628,179.561,5.980,149.201
C06565=1160.307,-26.460,-45.640,179.563,5.980,149.201
C06566=1160.302,-26.211,-45.653,179.565,5.981,149.200
C06567=1160.296,-25.961,-45.665,179.568,5.981,149.199
C06568=1160.291,-25.712,-45.677,179.570,5.982,149.199
C06569=1160.286,-25.462,-45.689,179.573,5.983,149.198
C06570=1160.281,-25.212,-45.702,179.575,5.983,149.198
C06571=1160.275,-24.962,-45.714,179.577,5.984,149.197
C06572=1160.271,-24.713,-45.726,179.580,5.984,149.196
C06573=1160.265,-24.443,-45.739,179.582,5.985,149.196
C06574=1160.260,-24.173,-45.753,179.585,5.985,149.195
C06575=1160.254,-23.903,-45.766,179.588,5.986,149.195
C06576=1160.248,-23.633,-45.780,179.591,5.987,149.194
C06577=1160.243,-23.383,-45.792,179.593,5.988,149.193
C06578=1160.238,-23.134,-45.804,179.596,5.988,149.193
C06579=1160.232,-22.884,-45.816,179.597,5.988,149.192
C06580=1160.227,-22.635,-45.829,179.600,5.989,149.192
C06581=1160.223,-22.385,-45.842,179.602,5.990,149.191
C06582=1160.217,-22.135,-45.854,179.605,5.990,149.190
C06583=1160.212,-21.885,-45.866,179.607,5.991,149.190
C06584=1160.207,-21.636,-45.879,179.610,5.991,149.189
C06585=1160.201,-21.386,-45.891,179.612,5.992,149.189
C06586=1160.196,-21.137,-45.903,179.614,5.993,149.188
C06587=1160.191,-20.888,-45.916,179.617,5.993,149.187
C06588=1160.186,-20.637,-45.928,179.619,5.994,149.187
C06589=1160.181,-20.388,-45.941,179.622,5.994,149.186
C06590=1160.176,-20.138,-45.953,179.624,5.995,149.186
C06591=1160.171,-19.889,-45.966,179.627,5.995,149.185
C06592=1160.166,-19.639,-45.978,179.629,5.996,149.185
C06593=1160.160,-19.390,-45.991,179.632,5.997,149.184
C06594=1160.155,-19.139,-46.004,179.634,5.997,149.183
C06595=1160.150,-18.889,-46.016,179.636,5.998,149.183
C06596=1160.145,-18.640,-46.029,179.639,5.999,149.182
C06597=1160.140,-18.391,-46.041,179.641,5.999,149.182
C06598=1160.134,-18.141,-46.054,179.644,6.000,149.181
C06599=1160.129,-17.892,-46.066,179.646,6.000,149.180
C06600=1160.124,-17.642,-46.079,179.649,6.001,149.180
C06601=1160.119,-17.392,-46.091,179.651,6.002,149.179
C06602=1160.113,-17.143,-46.104,179.654,6.002,149.178
C06603=1160.108,-16.893,-46.117,179.656,6.003,149.178
C06604=1160.104,-16.643,-46.130,179.658,6.003,149.177
C06605=1160.098,-16.393,-46.142,179.661,6.004,149.177
C06606=1160.093,-16.144,-46.155,179.663,6.005,149.176
C06607=1160.088,-15.895,-46.167,179.665,6.005,149.176
C06608=1160.083,-15.645,-46.180,179.668,6.006,149.175
C06609=1160.078,-15.395,-46.193,179.671,6.006,149.174
C06610=1160.073,-15.146,-46.206,179.673,6.007,149.174
C06611=1160.068,-14.896,-46.218,179.676,6.008,149.173
C06612=1160.062,-14.646,-46.230,179.678,6.008,149.173
C06613=1160.058,-14.396,-46.243,179.680,6.009,149.172
C06614=1160.052,-14.147,-46.257,179.683,6.010,149.172
C06615=1160.047,-13.897,-46.269,179.685,6.010,149.171
C06616=1160.041,-13.648,-46.282,179.687,6.011,149.170
C06617=1160.037,-13.398,-46.295,179.690,6.011,149.170
C06618=1160.031,-13.149,-46.308,179.692,6.012,149.169
C06619=1160.026,-12.899,-46.321,179.695,6.013,149.169
C06620=1160.021,-12.649,-46.333,179.697,6.013,149.168
C06621=1160.016,-12.400,-46.346,179.700,6.014,149.167
C06622=1160.011,-12.151,-46.359,179.702,6.014,149.167
C06623=1160.005,-11.901,-46.372,179.705,6.015,149.166
C06624=1160.001,-11.651,-46.385,179.707,6.015,149.165
C06625=1159.996,-11.402,-46.397,179.709,6.016,149.165
C06626=1159.990,-11.152,-46.411,179.712,6.017,149.164
C06627=1159.985,-10.902,-46.424,179.714,6.018,149.164
C06628=1159.980,-10.653,-46.436,179.717,6.018,149.163
C06629=1159.975,-10.403,-46.449,179.719,6.019,149.163
C06630=1159.970,-10.153,-46.462,179.722,6.020,149.162
C06631=1159.965,-9.904,-46.475,179.725,6.021,149.162
C06632=1159.960,-9.654,-46.488,179.727,6.021,149.161
C06633=1159.954,-9.404,-46.501,179.730,6.022,149.160
C06634=1159.949,-9.155,-46.514,179.732,6.023,149.160
C06635=1159.944,-8.905,-46.526,179.735,6.023,149.159
C06636=1159.939,-8.655,-46.540,179.737,6.024,149.159
C06637=1159.934,-8.406,-46.552,179.740,6.024,149.158
C06638=1159.929,-8.156,-46.565,179.742,6.025,149.157
C06639=1159.923,-7.906,-46.579,179.744,6.026,149.157
C06640=1159.918,-7.657,-46.592,179.747,6.026,149.156
C06641=1159.913,-7.408,-46.605,179.749,6.027,149.156
C06642=1159.908,-7.158,-46.618,179.751,6.028,149.155
C06643=1159.903,-6.908,-46.631,179.754,6.028,149.154
C06644=1159.898,-6.659,-46.643,179.756,6.029,149.154
C06645=1159.893,-6.409,-46.657,179.759,6.029,149.153
C06646=1159.887,-6.159,-46.669,179.762,6.030,149.153
C06647=1159.882,-5.910,-46.684,179.764,6.031,149.152
C06648=1159.877,-5.660,-46.696,179.766,6.031,149.151
C06649=1159.872,-5.411,-46.709,179.769,6.032,149.151
C06650=1159.867,-5.161,-46.723,179.772,6.033,149.150
C06651=1159.862,-4.911,-46.735,179.774,6.034,149.150
C06652=1159.857,-4.662,-46.749,179.777,6.034,149.149
C06653=1159.852,-4.412,-46.762,179.779,6.035,149.149
C06654=1159.846,-4.163,-46.775,179.781,6.036,149.148
C06655=1159.841,-3.913,-46.788,179.784,6.036,149.147
C06656=1159.836,-3.664,-46.802,179.786,6.037,149.147
C06657=1159.831,-3.414,-46.815,179.789,6.037,149.146
C06658=1159.826,-3.164,-46.828,179.791,6.038,149.146
C06659=1159.820,-2.915,-46.841,179.794,6.039,149.145
C06660=1159.816,-2.665,-46.855,179.796,6.039,149.144
C06661=1159.810,-2.416,-46.868,179.799,6.040,149.144
C06662=1159.806,-2.166,-46.881,179.801,6.041,149.143
C06663=1159.800,-1.917,-46.895,179.804,6.042,149.143
C06664=1159.796,-1.667,-46.908,179.806,6.043,149.142
C06665=1159.790,-1.417,-46.921,179.809,6.043,149.141
C06666=1159.786,-1.168,-46.934,179.811,6.044,149.141
C06667=1159.780,-0.918,-46.948,179.814,6.044,149.140
C06668=1159.775,-0.668,-46.961,179.816,6.045,149.140
C06669=1159.770,-0.419,-46.975,179.819,6.046,149.139
C06670=1159.764,-0.169,-46.988,179.821,6.046,149.138
C06671=1159.759,0.081,-47.001,179.823,6.047,149.138
C06672=1159.754,0.330,-47.015,179.826,6.047,149.137
C06673=1159.749,0.580,-47.028,179.828,6.048,149.137
C06674=1159.744,0.829,-47.041,179.831,6.049,149.136
C06675=1159.739,1.079,-47.054,179.834,6.050,149.136
C06676=1159.733,1.328,-47.068,179.836,6.051,149.135
C06677=1159.728,1.598,-47.083,179.839,6.051,149.134
C06678=1159.723,1.867,-47.097,179.841,6.052,149.134
C06679=1159.717,2.137,-47.111,179.844,6.053,149.133
C06680=1159.711,2.406,-47.126,179.847,6.054,149.132
C06681=1159.706,2.655,-47.140,179.849,6.055,149.132
C06682=1159.701,2.905,-47.153,179.852,6.055,149.131
C06683=1159.696,3.155,-47.166,179.854,6.056,149.131
C06684=1159.691,3.404,-47.180,179.857,6.056,149.130
C06685=1159.686,3.654,-47.193,179.859,6.057,149.130
C06686=1159.681,3.904,-47.208,179.862,6.058,149.129
C06687=1159.676,4.153,-47.220,179.864,6.059,149.129
C06688=1159.671,4.403,-47.234,179.867,6.060,149.128
C06689=1159.665,4.652,-47.248,179.870,6.060,149.127
C06690=1159.661,4.902,-47.261,179.872,6.061,149.127
C06691=1159.655,5.151,-47.275,179.874,6.061,149.126
C06692=1159.650,5.401,-47.289,179.877,6.062,149.126
C06693=1159.645,5.650,-47.302,179.879,6.063,149.125
C06694=1159.640,5.900,-47.316,179.882,6.064,149.124
C06695=1159.635,6.150,-47.330,179.885,6.065,149.124
C06696=1159.630,6.399,-47.343,179.887,6.066,149.123
C06697=1159.625,6.649,-47.357,179.889,6.066,149.123
C06698=1159.619,6.898,-47.371,179.892,6.067,149.122
C06699=1159.615,7.148,-47.384,179.894,6.067,149.121
C06700=1159.610,7.398,-47.398,179.896,6.068,149.121
C06701=1159.604,7.647,-47.412,179.899,6.069,149.120
C06702=1159.599,7.897,-47.425,179.902,6.070,149.120
C06703=1159.594,8.146,-47.439,179.905,6.071,149.119
C06704=1159.589,8.395,-47.453,179.907,6.071,149.118
C06705=1159.584,8.646,-47.467,179.909,6.072,149.118
C06706=1159.578,8.895,-47.480,179.912,6.072,149.117
C06707=1159.574,9.144,-47.494,179.914,6.073,149.117
C06708=1159.568,9.394,-47.507,179.917,6.074,149.116
C06709=1159.563,9.643,-47.522,179.920,6.075,149.116
C06710=1159.558,9.893,-47.536,179.922,6.076,149.115
C06711=1159.553,10.142,-47.549,179.924,6.077,149.115
C06712=1159.548,10.392,-47.563,179.927,6.077,149.114
C06713=1159.543,10.642,-47.577,179.929,6.078,149.113
C06714=1159.538,10.891,-47.591,179.932,6.078,149.113
C06715=1159.533,11.141,-47.605,179.935,6.080,149.112
C06716=1159.528,11.391,-47.619,179.937,6.080,149.112
C06717=1159.523,11.640,-47.632,179.940,6.081,149.111
C06718=1159.518,11.889,-47.646,179.942,6.082,149.110
C06719=1159.513,12.140,-47.660,179.945,6.082,149.110
C06720=1159.507,12.389,-47.674,179.947,6.083,149.109
C06721=1159.502,12.638,-47.688,179.950,6.084,149.109
C06722=1159.497,12.888,-47.702,179.952,6.085,149.108
C06723=1159.492,13.137,-47.716,179.955,6.086,149.107
C06724=1159.487,13.386,-47.730,179.957,6.086,149.107
C06725=1159.482,13.637,-47.744,179.960,6.087,149.106
C06726=1159.477,13.886,-47.758,179.962,6.088,149.106
C06727=1159.472,14.135,-47.772,179.965,6.089,149.105
C06728=1159.467,14.385,-47.786,179.967,6.090,149.105
C06729=1159.462,14.635,-47.800,179.970,6.090,149.104
C06730=1159.456,14.884,-47.814,179.972,6.091,149.104
C06731=1159.451,15.134,-47.829,179.975,6.092,149.103
C06732=1159.447,15.384,-47.841,179.978,6.093,149.102
C06733=1159.441,15.633,-47.855,179.980,6.094,149.102
C06734=1159.436,15.882,-47.870,179.982,6.094,149.101
C06735=1159.431,16.132,-47.884,179.985,6.095,149.101
C06736=1159.426,16.382,-47.898,179.988,6.095,149.100
C06737=1159.421,16.631,-47.912,179.990,6.097,149.100
C06738=1159.416,16.881,-47.926,179.993,6.097,149.099
C06739=1159.411,17.130,-47.941,179.995,6.098,149.098
C06740=1159.406,17.380,-47.955,179.998,6.099,149.098
C06741=1159.400,17.629,-47.969,-180.000,6.100,149.097
C06742=1159.395,17.879,-47.983,-179.997,6.101,149.097
C06743=1159.390,18.128,-47.997,-179.994,6.102,149.096
C06744=1159.385,18.378,-48.012,-179.992,6.102,149.095
C06745=1159.380,18.628,-48.026,-179.990,6.103,149.095
C06746=1159.375,18.877,-48.040,-179.987,6.103,149.094
C06747=1159.370,19.127,-48.054,-179.984,6.105,149.094
C06748=1159.365,19.376,-48.068,-179.982,6.106,149.093
C06749=1159.360,19.626,-48.083,-179.979,6.106,149.093
C06750=1159.354,19.875,-48.097,-179.977,6.107,149.092
C06751=1159.349,20.125,-48.111,-179.975,6.108,149.092
C06752=1159.345,20.374,-48.125,-179.971,6.109,149.091
C06753=1159.340,20.624,-48.139,-179.969,6.110,149.090
C06754=1159.335,20.873,-48.154,-179.967,6.110,149.090
C06755=1159.330,21.123,-48.169,-179.964,6.111,149.089
C06756=1159.324,21.372,-48.183,-179.962,6.112,149.089
C06757=1159.319,21.622,-48.197,-179.959,6.113,149.088
C06758=1159.314,21.871,-48.211,-179.956,6.114,149.087
C06759=1159.310,22.121,-48.225,-179.954,6.114,149.087
C06760=1159.304,22.371,-48.240,-179.952,6.115,149.086
C06761=1159.299,22.621,-48.255,-179.948,6.116,149.086
C06762=1159.294,22.869,-48.269,-179.946,6.117,149.085
C06763=1159.289,23.119,-48.284,-179.943,6.118,149.085
C06764=1159.284,23.369,-48.298,-179.941,6.118,149.084
C06765=1159.279,23.618,-48.312,-179.938,6.120,149.083
C06766=1159.274,23.868,-48.326,-179.936,6.120,149.083
C06767=1159.269,24.117,-48.341,-179.933,6.121,149.082
C06768=1159.264,24.367,-48.356,-179.931,6.122,149.082
C06769=1159.258,24.616,-48.370,-179.928,6.123,149.081
C06770=1159.253,24.866,-48.384,-179.926,6.124,149.081
C06771=1159.248,25.116,-48.399,-179.923,6.124,149.080
C06772=1159.243,25.365,-48.414,-179.921,6.125,149.080
C06773=1159.238,25.614,-48.428,-179.918,6.126,149.079
C06774=1159.233,25.864,-48.442,-179.915,6.127,149.078
C06775=1159.228,26.113,-48.458,-179.913,6.128,149.078
C06776=1159.223,26.363,-48.472,-179.911,6.129,149.077
C06777=1159.218,26.613,-48.486,-179.907,6.130,149.077
C06778=1159.213,26.863,-48.501,-179.905,6.131,149.076
C06779=1159.208,27.111,-48.515,-179.903,6.131,149.075
C06780=1159.202,27.361,-48.530,-179.900,6.132,149.075
C06781=1159.197,27.630,-48.546,-179.897,6.133,149.074
C06782=1159.192,27.899,-48.562,-179.895,6.134,149.074
C06783=1159.187,28.167,-48.577,-179.892,6.135,149.073
C06784=1159.181,28.436,-48.594,-179.889,6.136,149.073
C06785=1159.176,28.686,-48.608,-179.886,6.136,149.072
C06786=1159.171,28.936,-48.622,-179.884,6.138,149.071
C06787=1159.166,29.185,-48.638,-179.881,6.138,149.071
C06788=1159.161,29.435,-48.652,-179.879,6.139,149.070
C06789=1159.156,29.684,-48.667,-179.876,6.140,149.070
C06790=1159.151,29.934,-48.681,-179.874,6.141,149.069
C06791=1159.145,30.184,-48.696,-179.871,6.142,149.068
C06792=1159.141,30.433,-48.711,-179.869,6.143,149.068
C06793=1159.136,30.683,-48.725,-179.865,6.144,149.067
C06794=1159.130,30.932,-48.741,-179.863,6.145,149.067
C06795=1159.126,31.182,-48.755,-179.861,6.145,149.066
C06796=1159.121,31.431,-48.770,-179.858,6.146,149.066
C06797=1159.116,31.681,-48.785,-179.855,6.147,149.065
C06798=1159.111,31.930,-48.800,-179.853,6.148,149.065
C06799=1159.106,32.180,-48.814,-179.850,6.149,149.064
C06800=1159.101,32.429,-48.829,-179.848,6.150,149.063
C06801=1159.095,32.679,-48.844,-179.845,6.151,149.063
C06802=1159.091,32.928,-48.859,-179.843,6.152,149.062
C06803=1159.085,33.178,-48.874,-179.840,6.152,149.062
C06804=1159.080,33.427,-48.889,-179.837,6.154,149.061
C06805=1159.075,33.677,-48.903,-179.835,6.154,149.061
C06806=1159.070,33.926,-48.919,-179.833,6.155,149.060
C06807=1159.065,34.176,-48.933,-179.829,6.156,149.059
C06808=1159.060,34.425,-48.948,-179.827,6.157,149.059
C06809=1159.055,34.674,-48.964,-179.825,6.158,149.058
C06810=1159.050,34.924,-48.978,-179.822,6.159,149.058
C06811=1159.045,35.173,-48.994,-179.819,6.160,149.057
C06812=1159.040,35.423,-49.008,-179.817,6.161,149.057
C06813=1159.035,35.672,-49.023,-179.814,6.162,149.056
C06814=1159.030,35.922,-49.039,-179.812,6.163,149.056
C06815=1159.025,36.171,-49.053,-179.809,6.163,149.055
C06816=1159.019,36.421,-49.068,-179.806,6.165,149.054
C06817=1159.015,36.670,-49.083,-179.804,6.165,149.054
C06818=1159.009,36.921,-49.099,-179.801,6.166,149.053
C06819=1159.005,37.170,-49.114,-179.799,6.167,149.053
C06820=1158.999,37.419,-49.129,-179.796,6.168,149.052
C06821=1158.995,37.669,-49.144,-179.794,6.169,149.052
C06822=1158.989,37.918,-49.159,-179.791,6.170,149.051
C06823=1158.984,38.167,-49.174,-179.789,6.171,149.051
C06824=1158.979,38.417,-49.190,-179.786,6.172,149.050
C06825=1158.974,38.666,-49.204,-179.784,6.173,149.050
C06826=1158.969,38.916,-49.220,-179.780,6.174,149.049
C06827=1158.964,39.165,-49.235,-179.778,6.175,149.048
C06828=1158.959,39.415,-49.251,-179.776,6.175,149.048
C06829=1158.954,39.665,-49.265,-179.773,6.177,149.047
C06830=1158.949,39.914,-49.280,-179.770,6.177,149.047
C06831=1158.944,40.163,-49.295,-179.768,6.178,149.046
C06832=1158.939,40.413,-49.311,-179.765,6.180,149.046
C06833=1158.934,40.662,-49.325,-179.763,6.180,149.045
C06834=1158.929,40.912,-49.341,-179.760,6.182,149.044
C06835=1158.924,41.162,-49.357,-179.757,6.183,149.044
C06836=1158.919,41.411,-49.372,-179.755,6.183,149.043
C06837=1158.914,41.660,-49.387,-179.752,6.185,149.043
C06838=1158.909,41.909,-49.402,-179.749,6.185,149.042
C06839=1158.904,42.159,-49.418,-179.747,6.186,149.042
C06840=1158.899,42.408,-49.432,-179.744,6.187,149.041
C06841=1158.894,42.659,-49.448,-179.742,6.188,149.041
C06842=1158.889,42.908,-49.464,-179.739,6.189,149.040
C06843=1158.884,43.157,-49.479,-179.736,6.190,149.039
C06844=1158.879,43.406,-49.494,-179.734,6.191,149.039
C06845=1158.873,43.656,-49.510,-179.732,6.192,149.038
C06846=1158.869,43.906,-49.525,-179.729,6.193,149.038
C06847=1158.864,44.155,-49.541,-179.726,6.194,149.037
C06848=1158.859,44.404,-49.556,-179.723,6.195,149.037
C06849=1158.854,44.654,-49.571,-179.721,6.196,149.036
C06850=1158.848,44.903,-49.587,-179.719,6.197,149.036
C06851=1158.844,45.153,-49.602,-179.715,6.198,149.035
C06852=1158.839,45.402,-49.618,-179.713,6.199,149.035
C06853=1158.833,45.652,-49.634,-179.711,6.199,149.034
C06854=1158.829,45.901,-49.649,-179.708,6.201,149.033
C06855=1158.824,46.151,-49.665,-179.705,6.202,149.033
C06856=1158.819,46.400,-49.680,-179.702,6.203,149.032
C06857=1158.813,46.650,-49.696,-179.700,6.204,149.032
C06858=1158.809,46.899,-49.711,-179.698,6.205,149.031
C06859=1158.804,47.149,-49.727,-179.694,6.206,149.031
C06860=1158.798,47.398,-49.742,-179.692,6.207,149.030
C06861=1158.794,47.647,-49.757,-179.690,6.208,149.030
C06862=1158.788,47.897,-49.773,-179.687,6.209,149.029
C06863=1158.784,48.147,-49.789,-179.685,6.210,149.029
C06864=1158.778,48.396,-49.804,-179.681,6.211,149.028
C06865=1158.774,48.645,-49.819,-179.679,6.212,149.027
C06866=1158.769,48.895,-49.835,-179.676,6.213,149.027
C06867=1158.764,49.144,-49.852,-179.674,6.214,149.026
C06868=1158.758,49.394,-49.867,-179.671,6.214,149.026
C06869=1158.754,49.643,-49.882,-179.669,6.216,149.025
C06870=1158.749,49.893,-49.898,-179.666,6.217,149.025
C06871=1158.744,50.142,-49.914,-179.663,6.218,149.024
C06872=1158.738,50.392,-49.929,-179.661,6.219,149.024
C06873=1158.733,50.642,-49.945,-179.658,6.220,149.023
C06874=1158.729,50.890,-49.961,-179.656,6.221,149.023
C06875=1158.724,51.139,-49.977,-179.653,6.222,149.022
C06876=1158.719,51.390,-49.993,-179.650,6.223,149.021
C06877=1158.713,51.639,-50.008,-179.648,6.224,149.021
C06878=1158.708,51.888,-50.024,-179.645,6.225,149.020
C06879=1158.704,52.138,-50.040,-179.642,6.226,149.020
C06880=1158.699,52.387,-50.055,-179.640,6.227,149.019
C06881=1158.694,52.637,-50.071,-179.637,6.228,149.019
C06882=1158.689,52.886,-50.088,-179.635,6.229,149.018
C06883=1158.684,53.135,-50.103,-179.632,6.231,149.018
C06884=1158.679,53.385,-50.119,-179.629,6.231,149.017
C06885=1158.673,53.654,-50.136,-179.626,6.233,149.016
C06886=1158.668,53.922,-50.153,-179.624,6.233,149.016
C06887=1158.662,54.191,-50.170,-179.621,6.235,149.015
C06888=1158.657,54.459,-50.187,-179.619,6.236,149.015
C06889=1158.652,54.709,-50.204,-179.615,6.237,149.014
C06890=1158.647,54.958,-50.219,-179.613,6.238,149.014
C06891=1158.642,55.208,-50.235,-179.610,6.239,149.013
C06892=1158.637,55.457,-50.252,-179.608,6.240,149.013
C06893=1158.632,55.706,-50.267,-179.605,6.241,149.012
C06894=1158.628,55.956,-50.283,-179.602,6.242,149.011
C06895=1158.622,56.205,-50.299,-179.600,6.244,149.011
C06896=1158.618,56.455,-50.315,-179.597,6.244,149.010
C06897=1158.613,56.704,-50.331,-179.595,6.245,149.010
C06898=1158.608,56.954,-50.347,-179.592,6.246,149.009
C06899=1158.603,57.203,-50.364,-179.589,6.247,149.009
C06900=1158.597,57.452,-50.379,-179.586,6.248,149.008
C06901=1158.593,57.702,-50.395,-179.584,6.249,149.008
C06902=1158.587,57.951,-50.411,-179.581,6.251,149.007
C06903=1158.583,58.201,-50.427,-179.579,6.252,149.007
C06904=1158.578,58.450,-50.444,-179.576,6.253,149.006
C06905=1158.573,58.700,-50.460,-179.573,6.254,149.006
C06906=1158.568,58.949,-50.476,-179.571,6.255,149.005
C06907=1158.563,59.199,-50.492,-179.568,6.256,149.004
C06908=1158.557,59.448,-50.509,-179.565,6.258,149.004
C06909=1158.552,59.698,-50.525,-179.563,6.258,149.004
C06910=1158.547,59.947,-50.541,-179.560,6.259,149.003
C06911=1158.542,60.196,-50.557,-179.558,6.261,149.002
C06912=1158.537,60.446,-50.573,-179.555,6.261,149.002
C06913=1158.532,60.695,-50.590,-179.552,6.263,149.001
C06914=1158.527,60.945,-50.605,-179.550,6.263,149.001
C06915=1158.522,61.194,-50.622,-179.547,6.265,149.000
C06916=1158.518,61.444,-50.638,-179.545,6.266,149.000
C06917=1158.513,61.692,-50.654,-179.542,6.267,148.999
C06918=1158.508,61.942,-50.671,-179.539,6.268,148.999
C06919=1158.503,62.192,-50.687,-179.536,6.269,148.998
C06920=1158.497,62.441,-50.704,-179.534,6.270,148.998
C06921=1158.493,62.691,-50.720,-179.531,6.271,148.997
C06922=1158.488,62.940,-50.736,-179.529,6.272,148.997
C06923=1158.483,63.189,-50.753,-179.526,6.274,148.996
C06924=1158.478,63.439,-50.768,-179.523,6.274,148.995
C06925=1158.473,63.688,-50.785,-179.521,6.276,148.995
C06926=1158.468,63.937,-50.801,-179.518,6.277,148.994
C06927=1158.463,64.188,-50.818,-179.515,6.278,148.994
C06928=1158.458,64.436,-50.834,-179.513,6.279,148.993
C06929=1158.453,64.686,-50.851,-179.510,6.280,148.993
C06930=1158.449,64.935,-50.867,-179.508,6.281,148.992
C06931=1158.443,65.185,-50.883,-179.504,6.283,148.992
C06932=1158.439,65.434,-50.900,-179.502,6.283,148.991
C06933=1158.433,65.683,-50.916,-179.500,6.285,148.991
C06934=1158.428,65.933,-50.933,-179.497,6.286,148.990
C06935=1158.424,66.183,-50.949,-179.494,6.287,148.990
C06936=1158.419,66.432,-50.965,-179.491,6.288,148.989
C06937=1158.413,66.681,-50.983,-179.489,6.289,148.989
C06938=1158.408,66.930,-50.999,-179.487,6.290,148.988
C06939=1158.404,67.180,-51.016,-179.483,6.292,148.988
C06940=1158.399,67.430,-51.032,-179.481,6.293,148.987
C06941=1158.393,67.679,-51.048,-179.478,6.294,148.986
C06942=1158.389,67.928,-51.065,-179.476,6.295,148.986
C06943=1158.384,68.177,-51.081,-179.473,6.296,148.986
C06944=1158.379,68.427,-51.098,-179.470,6.298,148.985
C06945=1158.374,68.676,-51.115,-179.468,6.299,148.984
C06946=1158.369,68.925,-51.132,-179.465,6.300,148.984
C06947=1158.364,69.175,-51.148,-179.462,6.301,148.983
C06948=1158.359,69.425,-51.165,-179.460,6.302,148.983
C06949=1158.354,69.674,-51.181,-179.457,6.303,148.982
C06950=1158.349,69.923,-51.198,-179.454,6.305,148.982
C06951=1158.344,70.173,-51.215,-179.452,6.305,148.981
C06952=1158.339,70.422,-51.231,-179.449,6.307,148.981
C06953=1158.335,70.671,-51.248,-179.447,6.308,148.980
C06954=1158.329,70.921,-51.265,-179.444,6.309,148.980
C06955=1158.324,71.170,-51.282,-179.441,6.310,148.979
C06956=1158.320,71.420,-51.298,-179.438,6.311,148.979
C06957=1158.315,71.669,-51.316,-179.435,6.313,148.978
C06958=1158.309,71.918,-51.332,-179.433,6.314,148.978
C06959=1158.305,72.168,-51.349,-179.430,6.315,148.977
C06960=1158.300,72.417,-51.366,-179.428,6.316,148.977
C06961=1158.295,72.667,-51.382,-179.425,6.317,148.976
C06962=1158.289,72.916,-51.399,-179.423,6.318,148.976
C06963=1158.285,73.165,-51.416,-179.420,6.320,148.975
C06964=1158.280,73.415,-51.433,-179.417,6.321,148.974
C06965=1158.275,73.664,-51.450,-179.414,6.322,148.974
C06966=1158.270,73.914,-51.466,-179.412,6.324,148.974
C06967=1158.265,74.163,-51.484,-179.409,6.324,148.973
C06968=1158.261,74.412,-51.501,-179.406,6.326,148.973
C06969=1158.255,74.661,-51.518,-179.404,6.327,148.972
C06970=1158.250,74.911,-51.534,-179.401,6.328,148.971
C06971=1158.245,75.161,-51.552,-179.398,6.330,148.971
C06972=1158.241,75.410,-51.568,-179.396,6.330,148.970
C06973=1158.235,75.659,-51.585,-179.393,6.332,148.970
C06974=1158.230,75.909,-51.602,-179.391,6.333,148.970
C06975=1158.226,76.158,-51.620,-179.387,6.334,148.969
C06976=1158.221,76.407,-51.637,-179.385,6.335,148.968
C06977=1158.215,76.656,-51.654,-179.383,6.337,148.968
C06978=1158.211,76.906,-51.670,-179.379,6.338,148.967
C06979=1158.206,77.156,-51.687,-179.377,6.339,148.967
C06980=1158.201,77.404,-51.705,-179.375,6.340,148.966
C06981=1158.196,77.654,-51.722,-179.372,6.341,148.966
C06982=1158.191,77.903,-51.738,-179.369,6.343,148.965
C06983=1158.186,78.153,-51.756,-179.366,6.344,148.965
C06984=1158.182,78.402,-51.773,-179.364,6.345,148.964
C06985=1158.176,78.652,-51.790,-179.361,6.346,148.964
C06986=1158.171,78.901,-51.808,-179.358,6.347,148.963
C06987=1158.167,79.151,-51.824,-179.356,6.349,148.963
C06988=1158.161,79.399,-51.842,-179.353,6.350,148.962
C06989=1158.157,79.668,-51.860,-179.350,6.351,148.962
C06990=1158.151,79.937,-51.879,-179.348,6.353,148.961
C06991=1158.145,80.205,-51.897,-179.344,6.354,148.961
C06992=1158.141,80.473,-51.915,-179.342,6.356,148.960
C06993=1158.136,80.723,-51.933,-179.339,6.356,148.960
C06994=1158.130,80.972,-51.950,-179.336,6.358,148.959
C06995=1158.126,81.221,-51.968,-179.334,6.359,148.959
C06996=1158.120,81.470,-51.985,-179.331,6.360,148.958
C06997=1158.115,81.720,-52.002,-179.328,6.362,148.958
C06998=1158.111,81.969,-52.019,-179.325,6.363,148.957
C06999=1158.106,82.219,-52.037,-179.323,6.364,148.957
C07000=1158.101,82.468,-52.055,-179.320,6.365,148.956
C07001=1158.096,82.717,-52.071,-179.318,6.366,148.956
C07002=1158.091,82.967,-52.088,-179.315,6.368,148.955
C07003=1158.086,83.216,-52.106,-179.312,6.369,148.955
C07004=1158.081,83.465,-52.123,-179.310,6.370,148.954
C07005=1158.076,83.714,-52.141,-179.307,6.372,148.954
C07006=1158.071,83.964,-52.158,-179.304,6.373,148.953
C07007=1158.067,84.213,-52.175,-179.302,6.374,148.953
C07008=1158.062,84.463,-52.193,-179.299,6.375,148.952
C07009=1158.057,84.712,-52.211,-179.296,6.376,148.952
C07010=1158.052,84.962,-52.228,-179.294,6.378,148.951
C07011=1158.047,85.211,-52.245,-179.290,6.379,148.951
C07012=1158.042,85.461,-52.263,-179.288,6.380,148.950
C07013=1158.037,85.710,-52.281,-179.286,6.382,148.950
C07014=1158.032,85.959,-52.298,-179.282,6.383,148.949
C07015=1158.028,86.208,-52.315,-179.280,6.384,148.949
C07016=1158.023,86.458,-52.333,-179.277,6.386,148.948
C07017=1158.018,86.707,-52.350,-179.274,6.387,148.948
C07018=1158.013,86.956,-52.368,-179.272,6.388,148.947
C07019=1158.008,87.206,-52.386,-179.269,6.390,148.947
C07020=1158.003,87.455,-52.403,-179.266,6.391,148.946
C07021=1157.999,87.704,-52.421,-179.264,6.392,148.946
C07022=1157.993,87.954,-52.438,-179.261,6.394,148.945
C07023=1157.988,88.203,-52.456,-179.258,6.395,148.945
C07024=1157.984,88.452,-52.474,-179.256,6.396,148.944
C07025=1157.978,88.702,-52.492,-179.253,6.397,148.944
C07026=1157.974,88.951,-52.509,-179.250,6.399,148.943
C07027=1157.969,89.200,-52.527,-179.248,6.400,148.943
C07028=1157.964,89.449,-52.545,-179.245,6.401,148.942
C07029=1157.959,89.699,-52.562,-179.242,6.403,148.942
C07030=1157.954,89.948,-52.580,-179.240,6.404,148.941
C07031=1157.949,90.198,-52.598,-179.237,6.405,148.941
C07032=1157.944,90.447,-52.615,-179.234,6.407,148.940
C07033=1157.939,90.697,-52.633,-179.232,6.407,148.940
C07034=1157.935,90.945,-52.651,-179.229,6.409,148.939
C07035=1157.930,91.195,-52.669,-179.226,6.411,148.939
C07036=1157.925,91.444,-52.687,-179.224,6.411,148.938
C07037=1157.920,91.694,-52.704,-179.221,6.413,148.938
C07038=1157.915,91.943,-52.722,-179.218,6.415,148.937
C07039=1157.910,92.192,-52.740,-179.215,6.416,148.937
C07040=1157.905,92.441,-52.758,-179.213,6.417,148.936
C07041=1157.900,92.690,-52.776,-179.210,6.419,148.936
C07042=1157.895,92.940,-52.793,-179.207,6.420,148.935
C07043=1157.890,93.189,-52.811,-179.205,6.421,148.935
C07044=1157.885,93.438,-52.829,-179.202,6.423,148.934
C07045=1157.880,93.688,-52.847,-179.199,6.424,148.934
C07046=1157.876,93.938,-52.865,-179.197,6.425,148.934
C07047=1157.871,94.187,-52.883,-179.194,6.426,148.933
C07048=1157.866,94.436,-52.901,-179.191,6.428,148.933
C07049=1157.861,94.685,-52.919,-179.188,6.430,148.932
C07050=1157.856,94.934,-52.937,-179.186,6.430,148.931
C07051=1157.851,95.183,-52.955,-179.183,6.432,148.931
C07052=1157.846,95.433,-52.973,-179.180,6.434,148.931
C07053=1157.841,95.682,-52.991,-179.178,6.435,148.930
C07054=1157.836,95.932,-53.009,-179.175,6.436,148.930
C07055=1157.832,96.181,-53.027,-179.172,6.438,148.929
C07056=1157.827,96.431,-53.045,-179.170,6.439,148.929
C07057=1157.822,96.680,-53.063,-179.167,6.440,148.928
C07058=1157.817,96.929,-53.081,-179.164,6.442,148.928
C07059=1157.812,97.178,-53.099,-179.162,6.443,148.927
C07060=1157.807,97.428,-53.117,-179.159,6.445,148.927
C07061=1157.803,97.677,-53.136,-179.156,6.445,148.926
C07062=1157.798,97.926,-53.154,-179.153,6.447,148.926
C07063=1157.793,98.175,-53.172,-179.151,6.449,148.925
C07064=1157.788,98.424,-53.190,-179.148,6.451,148.925
C07065=1157.783,98.674,-53.208,-179.145,6.451,148.924
C07066=1157.778,98.923,-53.226,-179.143,6.453,148.924
C07067=1157.774,99.173,-53.245,-179.140,6.454,148.923
C07068=1157.768,99.422,-53.263,-179.138,6.455,148.923
C07069=1157.763,99.671,-53.281,-179.135,6.457,148.922
C07070=1157.758,99.920,-53.299,-179.132,6.458,148.922
C07071=1157.754,100.169,-53.318,-179.129,6.460,148.922
C07072=1157.750,100.419,-53.336,-179.127,6.461,148.921
C07073=1157.745,100.668,-53.354,-179.124,6.462,148.921
C07074=1157.739,100.918,-53.373,-179.121,6.464,148.920
C07075=1157.734,101.167,-53.391,-179.118,6.466,148.920
C07076=1157.730,101.417,-53.409,-179.115,6.467,148.919
C07077=1157.725,101.665,-53.428,-179.113,6.468,148.919
C07078=1157.720,101.914,-53.446,-179.110,6.470,148.918
C07079=1157.715,102.164,-53.464,-179.108,6.471,148.918
C07080=1157.710,102.414,-53.483,-179.105,6.473,148.917
C07081=1157.706,102.662,-53.501,-179.102,6.474,148.917
C07082=1157.701,102.911,-53.519,-179.099,6.475,148.916
C07083=1157.695,103.161,-53.538,-179.097,6.477,148.916
C07084=1157.691,103.411,-53.556,-179.094,6.479,148.916
C07085=1157.686,103.659,-53.575,-179.091,6.479,148.915
C07086=1157.681,103.909,-53.593,-179.089,6.481,148.914
C07087=1157.676,104.158,-53.612,-179.086,6.483,148.914
C07088=1157.672,104.407,-53.631,-179.083,6.484,148.914
C07089=1157.667,104.656,-53.649,-179.080,6.486,148.913
C07090=1157.661,104.906,-53.667,-179.078,6.487,148.913
C07091=1157.657,105.155,-53.686,-179.075,6.488,148.912
C07092=1157.652,105.404,-53.704,-179.072,6.490,148.912
C07093=1157.646,105.673,-53.724,-179.069,6.491,148.911
C07094=1157.642,105.941,-53.744,-179.067,6.493,148.911
C07095=1157.636,106.210,-53.765,-179.064,6.495,148.910
C07096=1157.631,106.478,-53.784,-179.061,6.496,148.910
C07097=1157.626,106.727,-53.803,-179.058,6.498,148.909
C07098=1157.622,106.977,-53.822,-179.055,6.499,148.909
C07099=1157.617,107.225,-53.840,-179.053,6.500,148.908
C07100=1157.611,107.475,-53.859,-179.050,6.502,148.908
C07101=1157.607,107.725,-53.877,-179.047,6.503,148.907
C07102=1157.602,107.973,-53.896,-179.044,6.505,148.907
C07103=1157.597,108.223,-53.915,-179.042,6.507,148.907
C07104=1157.593,108.472,-53.934,-179.039,6.507,148.906
C07105=1157.587,108.722,-53.952,-179.036,6.509,148.906
C07106=1157.583,108.970,-53.971,-179.034,6.511,148.905
C07107=1157.577,109.220,-53.990,-179.031,6.512,148.905
C07108=1157.573,109.469,-54.009,-179.028,6.514,148.904
C07109=1157.569,109.718,-54.028,-179.026,6.515,148.904
C07110=1157.563,109.968,-54.046,-179.023,6.516,148.903
C07111=1157.559,110.216,-54.065,-179.020,6.518,148.903
C07112=1157.554,110.466,-54.084,-179.017,6.520,148.902
C07113=1157.549,110.715,-54.103,-179.015,6.521,148.902
C07114=1157.544,110.965,-54.122,-179.011,6.523,148.901
C07115=1157.539,111.214,-54.140,-179.009,6.524,148.901
C07116=1157.534,111.462,-54.160,-179.007,6.525,148.901
C07117=1157.530,111.712,-54.178,-179.004,6.527,148.900
C07118=1157.524,111.961,-54.197,-179.001,6.529,148.900
C07119=1157.520,112.210,-54.216,-178.998,6.530,148.899
C07120=1157.515,112.460,-54.235,-178.995,6.532,148.899
C07121=1157.511,112.709,-54.254,-178.993,6.533,148.898
C07122=1157.505,112.958,-54.273,-178.990,6.534,148.898
C07123=1157.500,113.207,-54.291,-178.988,6.536,148.898
C07124=1157.496,113.457,-54.311,-178.984,6.538,148.897
C07125=1157.490,113.706,-54.330,-178.982,6.539,148.897
C07126=1157.486,113.956,-54.348,-178.979,6.541,148.896
C07127=1157.481,114.204,-54.368,-178.976,6.543,148.896
C07128=1157.477,114.454,-54.387,-178.974,6.544,148.895
C07129=1157.471,114.703,-54.406,-178.971,6.545,148.895
C07130=1157.466,114.953,-54.425,-178.968,6.547,148.894
C07131=1157.462,115.201,-54.444,-178.966,6.548,148.894
C07132=1157.457,115.451,-54.463,-178.963,6.550,148.893
C07133=1157.452,115.699,-54.482,-178.960,6.552,148.893
C07134=1157.448,115.949,-54.502,-178.957,6.553,148.893
C07135=1157.442,116.199,-54.520,-178.955,6.554,148.892
C07136=1157.438,116.448,-54.539,-178.952,6.556,148.892
C07137=1157.433,116.697,-54.559,-178.949,6.557,148.891
C07138=1157.428,116.946,-54.578,-178.947,6.559,148.891
C07139=1157.423,117.195,-54.597,-178.944,6.561,148.890
C07140=1157.418,117.444,-54.617,-178.941,6.562,148.890
C07141=1157.413,117.693,-54.636,-178.938,6.564,148.890
C07142=1157.409,117.942,-54.655,-178.935,6.566,148.889
C07143=1157.403,118.192,-54.674,-178.933,6.566,148.889
C07144=1157.399,118.442,-54.693,-178.930,6.568,148.888
C07145=1157.395,118.691,-54.712,-178.928,6.570,148.888
C07146=1157.389,118.940,-54.732,-178.925,6.572,148.887
C07147=1157.385,119.189,-54.751,-178.922,6.573,148.887
C07148=1157.379,119.438,-54.771,-178.919,6.575,148.886
C07149=1157.375,119.687,-54.790,-178.916,6.576,148.886
C07150=1157.370,119.936,-54.809,-178.914,6.578,148.886
C07151=1157.365,120.186,-54.829,-178.911,6.580,148.885
C07152=1157.360,120.435,-54.848,-178.909,6.581,148.885
C07153=1157.356,120.684,-54.867,-178.906,6.582,148.884
C07154=1157.351,120.933,-54.887,-178.903,6.584,148.884
C07155=1157.346,121.182,-54.906,-178.900,6.585,148.883
C07156=1157.341,121.432,-54.925,-178.897,6.587,148.883
C07157=1157.337,121.681,-54.945,-178.895,6.589,148.882
C07158=1157.332,121.930,-54.964,-178.892,6.591,148.882
C07159=1157.327,122.180,-54.983,-178.889,6.592,148.882
C07160=1157.322,122.429,-55.004,-178.887,6.594,148.881
C07161=1157.317,122.677,-55.023,-178.884,6.596,148.881
C07162=1157.312,122.927,-55.043,-178.882,6.597,148.880
C07163=1157.308,123.176,-55.061,-178.879,6.598,148.880
C07164=1157.303,123.425,-55.081,-178.876,6.600,148.879
C07165=1157.298,123.675,-55.101,-178.873,6.601,148.879
C07166=1157.293,123.924,-55.120,-178.870,6.603,148.879
C07167=1157.288,124.172,-55.140,-178.868,6.605,148.878
C07168=1157.284,124.422,-55.160,-178.865,6.607,148.878
C07169=1157.278,124.671,-55.179,-178.862,6.608,148.877
C07170=1157.274,124.920,-55.198,-178.860,6.610,148.877
C07171=1157.270,125.170,-55.218,-178.856,6.611,148.876
C07172=1157.265,125.419,-55.239,-178.854,6.613,148.876
C07173=1157.260,125.668,-55.258,-178.851,6.615,148.876
C07174=1157.255,125.917,-55.277,-178.848,6.616,148.875
C07175=1157.250,126.167,-55.297,-178.845,6.618,148.875
C07176=1157.245,126.415,-55.317,-178.843,6.619,148.874
C07177=1157.241,126.664,-55.337,-178.841,6.621,148.874
C07178=1157.236,126.914,-55.356,-178.838,6.623,148.874
C07179=1157.231,127.163,-55.376,-178.835,6.624,148.873
C07180=1157.226,127.412,-55.396,-178.832,6.626,148.873
C07181=1157.221,127.661,-55.416,-178.829,6.627,148.872
C07182=1157.217,127.911,-55.435,-178.827,6.629,148.872
C07183=1157.212,128.159,-55.455,-178.824,6.631,148.871
C07184=1157.207,128.409,-55.475,-178.821,6.632,148.871
C07185=1157.202,128.658,-55.495,-178.818,6.634,148.871
C07186=1157.198,128.907,-55.515,-178.816,6.636,148.870
C07187=1157.192,129.156,-55.534,-178.813,6.638,148.870
C07188=1157.188,129.405,-55.555,-178.810,6.639,148.869
C07189=1157.183,129.655,-55.574,-178.808,6.641,148.869
C07190=1157.178,129.904,-55.594,-178.805,6.643,148.869
C07191=1157.174,130.153,-55.614,-178.802,6.644,148.868
C07192=1157.169,130.402,-55.634,-178.799,6.646,148.868
C07193=1157.164,130.651,-55.654,-178.796,6.648,148.867
C07194=1157.159,130.901,-55.674,-178.794,6.649,148.867
C07195=1157.155,131.150,-55.694,-178.791,6.651,148.866
C07196=1157.150,131.398,-55.713,-178.788,6.653,148.866
C07197=1157.144,131.667,-55.736,-178.785,6.654,148.866
C07198=1157.139,131.935,-55.757,-178.783,6.656,148.865
C07199=1157.134,132.204,-55.779,-178.780,6.658,148.865
C07200=1157.129,132.472,-55.800,-178.776,6.660,148.864
C07201=1157.124,132.722,-55.820,-178.774,6.662,148.864
C07202=1157.120,132.971,-55.840,-178.771,6.663,148.864
C07203=1157.115,133.221,-55.860,-178.768,6.665,148.863
C07204=1157.110,133.470,-55.881,-178.765,6.667,148.863
C07205=1157.105,133.719,-55.901,-178.763,6.669,148.862
C07206=1157.100,133.968,-55.921,-178.760,6.670,148.862
C07207=1157.096,134.217,-55.941,-178.758,6.671,148.862
C07208=1157.091,134.466,-55.961,-178.755,6.673,148.861
C07209=1157.087,134.715,-55.981,-178.752,6.676,148.861
C07210=1157.081,134.964,-56.002,-178.749,6.677,148.860
C07211=1157.077,135.214,-56.022,-178.746,6.679,148.860
C07212=1157.072,135.463,-56.042,-178.744,6.681,148.860
C07213=1157.067,135.711,-56.062,-178.741,6.682,148.859
C07214=1157.062,135.961,-56.082,-178.738,6.684,148.859
C07215=1157.057,136.210,-56.103,-178.735,6.685,148.858
C07216=1157.053,136.459,-56.123,-178.732,6.687,148.858
C07217=1157.048,136.708,-56.143,-178.730,6.689,148.857
C07218=1157.044,136.957,-56.163,-178.727,6.691,148.857
C07219=1157.039,137.207,-56.184,-178.724,6.692,148.857
C07220=1157.034,137.456,-56.204,-178.722,6.694,148.856
C07221=1157.029,137.705,-56.224,-178.719,6.696,148.856
C07222=1157.024,137.954,-56.245,-178.716,6.698,148.855
C07223=1157.020,138.203,-56.265,-178.713,6.699,148.855
C07224=1157.015,138.452,-56.286,-178.711,6.701,148.855
C07225=1157.011,138.701,-56.306,-178.708,6.703,148.854
C07226=1157.005,138.950,-56.326,-178.705,6.704,148.854
C07227=1157.000,139.199,-56.346,-178.703,6.706,148.854
C07228=1156.996,139.448,-56.367,-178.700,6.708,148.853
C07229=1156.991,139.698,-56.388,-178.697,6.710,148.853
C07230=1156.986,139.947,-56.408,-178.694,6.711,148.852
C07231=1156.982,140.195,-56.429,-178.692,6.713,148.852
C07232=1156.977,140.445,-56.450,-178.689,6.715,148.852
C07233=1156.972,140.694,-56.469,-178.686,6.717,148.851
C07234=1156.967,140.944,-56.490,-178.684,6.718,148.851
C07235=1156.962,141.193,-56.510,-178.681,6.720,148.850
C07236=1156.958,141.441,-56.531,-178.678,6.722,148.850
C07237=1156.953,141.691,-56.552,-178.676,6.723,148.850
C07238=1156.948,141.940,-56.572,-178.673,6.725,148.849
C07239=1156.944,142.189,-56.593,-178.670,6.727,148.849
C07240=1156.939,142.438,-56.614,-178.667,6.729,148.848
C07241=1156.934,142.687,-56.634,-178.664,6.731,148.848
C07242=1156.929,142.936,-56.655,-178.661,6.733,148.848
C07243=1156.925,143.185,-56.675,-178.659,6.735,148.847
C07244=1156.919,143.434,-56.696,-178.656,6.736,148.847
C07245=1156.915,143.683,-56.717,-178.653,6.738,148.847
C07246=1156.910,143.933,-56.738,-178.651,6.740,148.846
C07247=1156.906,144.182,-56.758,-178.648,6.741,148.846
C07248=1156.902,144.431,-56.779,-178.645,6.743,148.845
C07249=1156.896,144.680,-56.800,-178.642,6.745,148.845
C07250=1156.892,144.929,-56.820,-178.640,6.747,148.845
C07251=1156.887,145.178,-56.842,-178.637,6.748,148.844
C07252=1156.883,145.427,-56.862,-178.634,6.750,148.844
C07253=1156.877,145.676,-56.883,-178.632,6.752,148.843
C07254=1156.873,145.925,-56.903,-178.629,6.754,148.843
C07255=1156.868,146.174,-56.924,-178.626,6.756,148.843
C07256=1156.863,146.424,-56.945,-178.623,6.758,148.842
C07257=1156.858,146.673,-56.966,-178.620,6.760,148.842
C07258=1156.853,146.921,-56.987,-178.618,6.761,148.842
C07259=1156.850,147.171,-57.008,-178.615,6.763,148.841
C07260=1156.844,147.420,-57.029,-178.612,6.765,148.841
C07261=1156.840,147.669,-57.049,-178.609,6.766,148.840
C07262=1156.835,147.918,-57.070,-178.607,6.768,148.840
C07263=1156.830,148.167,-57.092,-178.604,6.770,148.840
C07264=1156.825,148.416,-57.112,-178.601,6.772,148.839
C07265=1156.820,148.665,-57.133,-178.598,6.774,148.839
C07266=1156.816,148.914,-57.154,-178.595,6.776,148.839
C07267=1156.812,149.163,-57.176,-178.593,6.778,148.838
C07268=1156.806,149.413,-57.197,-178.590,6.780,148.838
C07269=1156.802,149.662,-57.217,-178.588,6.781,148.838
C07270=1156.797,149.910,-57.239,-178.585,6.783,148.837
C07271=1156.792,150.160,-57.260,-178.582,6.785,148.837
C07272=1156.787,150.409,-57.280,-178.580,6.787,148.836
C07273=1156.783,150.658,-57.302,-178.577,6.788,148.836
C07274=1156.778,150.907,-57.323,-178.574,6.791,148.836
C07275=1156.774,151.156,-57.344,-178.571,6.793,148.835
C07276=1156.769,151.405,-57.365,-178.568,6.794,148.835
C07277=1156.764,151.654,-57.386,-178.565,6.796,148.835
C07278=1156.760,151.903,-57.408,-178.563,6.798,148.834
C07279=1156.755,152.152,-57.429,-178.560,6.800,148.834
C07280=1156.750,152.402,-57.450,-178.557,6.801,148.833
C07281=1156.745,152.650,-57.471,-178.555,6.803,148.833
C07282=1156.740,152.899,-57.492,-178.551,6.806,148.833
C07283=1156.736,153.148,-57.514,-178.549,6.807,148.832
C07284=1156.731,153.398,-57.535,-178.546,6.809,148.832
C07285=1156.726,153.646,-57.556,-178.544,6.811,148.832
C07286=1156.722,153.895,-57.577,-178.541,6.813,148.831
C07287=1156.717,154.145,-57.599,-178.538,6.815,148.831
C07288=1156.712,154.394,-57.620,-178.536,6.816,148.831
C07289=1156.707,154.643,-57.641,-178.532,6.819,148.830
C07290=1156.702,154.892,-57.662,-178.530,6.821,148.830
C07291=1156.699,155.141,-57.684,-178.527,6.822,148.830
C07292=1156.694,155.389,-57.706,-178.524,6.824,148.829
C07293=1156.689,155.639,-57.727,-178.522,6.826,148.829
C07294=1156.684,155.887,-57.748,-178.519,6.828,148.828
C07295=1156.679,156.137,-57.770,-178.516,6.830,148.828
C07296=1156.674,156.386,-57.791,-178.513,6.832,148.828
C07297=1156.669,156.635,-57.813,-178.511,6.834,148.827
C07298=1156.666,156.884,-57.834,-178.508,6.836,148.827
C07299=1156.661,157.133,-57.855,-178.505,6.837,148.827
C07300=1156.655,157.382,-57.876,-178.503,6.839,148.826
C07301=1156.650,157.651,-57.900,-178.499,6.842,148.826
C07302=1156.646,157.920,-57.923,-178.497,6.843,148.826
C07303=1156.640,158.189,-57.947,-178.493,6.846,148.825
C07304=1156.636,158.458,-57.970,-178.491,6.848,148.825
C07305=1156.630,158.707,-57.991,-178.488,6.849,148.825
C07306=1156.626,158.956,-58.013,-178.485,6.851,148.824
C07307=1156.621,159.205,-58.035,-178.482,6.854,148.824
C07308=1156.616,159.454,-58.056,-178.479,6.855,148.823
C07309=1156.612,159.704,-58.078,-178.477,6.857,148.823
C07310=1156.607,159.952,-58.099,-178.474,6.859,148.823
C07311=1156.602,160.201,-58.121,-178.472,6.861,148.822
C07312=1156.598,160.450,-58.143,-178.468,6.864,148.822
C07313=1156.593,160.699,-58.165,-178.466,6.865,148.822
C07314=1156.588,160.949,-58.186,-178.463,6.867,148.821
C07315=1156.584,161.197,-58.208,-178.460,6.869,148.821
C07316=1156.579,161.446,-58.229,-178.458,6.871,148.821
C07317=1156.574,161.695,-58.252,-178.455,6.873,148.821
C07318=1156.570,161.944,-58.273,-178.452,6.875,148.820
C07319=1156.565,162.193,-58.295,-178.449,6.877,148.820
C07320=1156.560,162.442,-58.317,-178.447,6.879,148.819
C07321=1156.556,162.691,-58.339,-178.444,6.880,148.819
C07322=1156.551,162.941,-58.360,-178.441,6.883,148.819
C07323=1156.546,163.189,-58.382,-178.438,6.885,148.818
C07324=1156.542,163.439,-58.404,-178.436,6.887,148.818
C07325=1156.537,163.687,-58.425,-178.433,6.889,148.818
C07326=1156.533,163.937,-58.447,-178.430,6.891,148.817
C07327=1156.528,164.185,-58.469,-178.427,6.893,148.817
C07328=1156.523,164.434,-58.491,-178.424,6.895,148.817
C07329=1156.519,164.683,-58.513,-178.422,6.896,148.816
C07330=1156.513,164.932,-58.535,-178.419,6.898,148.816
C07331=1156.509,165.182,-58.557,-178.416,6.901,148.816
